LIN {X 0,Y 359.057,Z 1023.859,A -85,B 0,C 180,E1 26266.24,E2 26266.24} C_VEL
LIN {X 0,Y 361.976,Z 1017.878,A -85,B 0,C 180,E1 26267.168,E2 26267.168} C_VEL
LIN {X 0,Y 362.697,Z 1001.208,A -85,B 0,C 180,E1 26275.226,E2 26275.226} C_VEL
LIN {X 0,Y 363.155,Z 994.678,A -85,B 0,C 180,E1 26283.616,E2 26283.616} C_VEL
LIN {X 0,Y 361.753,Z 1005.173,A -85,B 0,C 180,E1 26293.358,E2 26293.358} C_VEL
LIN {X 0,Y 359.687,Z 1021.209,A -85,B 0,C 180,E1 26299.865,E2 26299.865} C_VEL
LIN {X 0,Y 316.249,Z 1080.703,A -85,B 0,C 180,E1 26305.848,E2 26305.848} C_VEL
LIN {X 0,Y 273.766,Z 1126.413,A -85,B 0,C 180,E1 26314.172,E2 26314.172} C_VEL
LIN {X 0,Y 249.213,Z 1145.042,A -85,B 0,C 180,E1 26318.032,E2 26318.032} C_VEL
LIN {X 0,Y 210.107,Z 1178.245,A -85,B 0,C 180,E1 26334.739,E2 26334.739} C_VEL
LIN {X 0,Y 190.164,Z 1197.047,A -85,B 0,C 180,E1 26356.165,E2 26356.165} C_VEL
LIN {X 0,Y 186.92,Z 1202.525,A -85,B 0,C 180,E1 26372.332,E2 26372.332} C_VEL
LIN {X 0,Y 188.619,Z 1200.708,A -85,B 0,C 180,E1 26392.237,E2 26392.237} C_VEL
LIN {X 0,Y 203.896,Z 1188.888,A -85,B 0,C 180,E1 26412.329,E2 26412.329} C_VEL
LIN {X 0,Y 242.392,Z 1161.787,A -85,B 0,C 180,E1 26431.043,E2 26431.043} C_VEL
LIN {X 0,Y 293.081,Z 1121.422,A -85,B 0,C 180,E1 26443.196,E2 26443.196} C_VEL
LIN {X 0,Y 345.638,Z 1068.573,A -85,B 0,C 180,E1 26450.834,E2 26450.834} C_VEL
LIN {X 0,Y 370.553,Z 1037.589,A -85,B 0,C 180,E1 26453.512,E2 26453.512} C_VEL
LIN {X 0,Y 372.422,Z 1029.57,A -85,B 0,C 180,E1 26461.144,E2 26461.144} C_VEL
LIN {X 0,Y 371.69,Z 1034.153,A -85,B 0,C 180,E1 26469.544,E2 26469.544} C_VEL
LIN {X 0,Y 369.889,Z 1039.513,A -85,B 0,C 180,E1 26472.259,E2 26472.259} C_VEL
LIN {X 0,Y 320.637,Z 1096.918,A -85,B 0,C 180,E1 26477.987,E2 26477.987} C_VEL
LIN {X 0,Y 267.811,Z 1144.547,A -85,B 0,C 180,E1 26487.487,E2 26487.487} C_VEL
LIN {X 0,Y 221.493,Z 1179.347,A -85,B 0,C 180,E1 26502.6,E2 26502.6} C_VEL
LIN {X 0,Y 193.031,Z 1200.435,A -85,B 0,C 180,E1 26524.393,E2 26524.393} C_VEL
LIN {X 0,Y 187.023,Z 1206.687,A -85,B 0,C 180,E1 26543.007,E2 26543.007} C_VEL
LIN {X 0,Y 187.02,Z 1205.903,A -85,B 0,C 180,E1 26556.979,E2 26556.979} C_VEL
LIN {X 0,Y 192.856,Z 1197.391,A -85,B 0,C 180,E1 26575.618,E2 26575.618} C_VEL
LIN {X 0,Y 218.915,Z 1173.79,A -85,B 0,C 180,E1 26596.656,E2 26596.656} C_VEL
LIN {X 0,Y 262.153,Z 1135.693,A -85,B 0,C 180,E1 26611.893,E2 26611.893} C_VEL
LIN {X 0,Y 311.561,Z 1084.366,A -85,B 0,C 180,E1 26621.632,E2 26621.632} C_VEL
LIN {X 0,Y 356.925,Z 1023.283,A -85,B 0,C 180,E1 26627.652,E2 26627.652} C_VEL
LIN {X 0,Y 358.203,Z 1006.363,A -85,B 0,C 180,E1 26636.382,E2 26636.382} C_VEL
LIN {X 0,Y 358.842,Z 1001.533,A -85,B 0,C 180,E1 26643.66,E2 26643.66} C_VEL
LIN {X 0,Y 357.045,Z 1012.278,A -85,B 0,C 180,E1 26653.538,E2 26653.538} C_VEL
LIN {X 0,Y 354.422,Z 1025.898,A -85,B 0,C 180,E1 26658.946,E2 26658.946} C_VEL
LIN {X 0,Y 308.073,Z 1086.636,A -85,B 0,C 180,E1 26665.255,E2 26665.255} C_VEL
LIN {X 0,Y 259.533,Z 1135.777,A -85,B 0,C 180,E1 26675.121,E2 26675.121} C_VEL
LIN {X 0,Y 249.213,Z 1145.042,A -85,B 0,C 180,E1 26678.032,E2 26678.032} C_VEL
LIN {X 0,Y 225.169,Z 1161.306,A -85,B 0,C 180,E1 26683.002,E2 26683.002} C_VEL
LIN {X 0,Y 192.438,Z 1187.662,A -85,B 0,C 180,E1 26701.79,E2 26701.79} C_VEL
LIN {X 0,Y 180.183,Z 1200.25,A -85,B 0,C 180,E1 26722.754,E2 26722.754} C_VEL
LIN {X 0,Y 178.43,Z 1202.977,A -85,B 0,C 180,E1 26737.331,E2 26737.331} C_VEL
LIN {X 0,Y 182.737,Z 1199.383,A -85,B 0,C 180,E1 26757.164,E2 26757.164} C_VEL
LIN {X 0,Y 205.467,Z 1183.588,A -85,B 0,C 180,E1 26779.28,E2 26779.28} C_VEL
LIN {X 0,Y 250.904,Z 1152.675,A -85,B 0,C 180,E1 26796.45,E2 26796.45} C_VEL
LIN {X 0,Y 305.086,Z 1108.368,A -85,B 0,C 180,E1 26807.14,E2 26807.14} C_VEL
LIN {X 0,Y 355.92,Z 1054.683,A -85,B 0,C 180,E1 26813.416,E2 26813.416} C_VEL
LIN {X 0,Y 365.792,Z 1042.038,A -85,B 0,C 180,E1 26814.623,E2 26814.623} C_VEL
LIN {X 0,Y 367.489,Z 1035.884,A -85,B 0,C 180,E1 26821.159,E2 26821.159} C_VEL
LIN {X 0,Y 366.523,Z 1040.357,A -85,B 0,C 180,E1 26829.505,E2 26829.505} C_VEL
LIN {X 0,Y 364.486,Z 1044.856,A -85,B 0,C 180,E1 26831.368,E2 26831.368} C_VEL
LIN {X 0,Y 314.252,Z 1101.025,A -85,B 0,C 180,E1 26837.107,E2 26837.107} C_VEL
LIN {X 0,Y 259.41,Z 1148.26,A -85,B 0,C 180,E1 26846.929,E2 26846.929} C_VEL
LIN {X 0,Y 212.09,Z 1181.955,A -85,B 0,C 180,E1 26862.744,E2 26862.744} C_VEL
LIN {X 0,Y 185.615,Z 1200.406,A -85,B 0,C 180,E1 26883.291,E2 26883.291} C_VEL
LIN {X 0,Y 179.014,Z 1206.607,A -85,B 0,C 180,E1 26902.693,E2 26902.693} C_VEL
LIN {X 0,Y 179.014,Z 1205.79,A -85,B 0,C 180,E1 26917.293,E2 26917.293} C_VEL
LIN {X 0,Y 185.425,Z 1197.223,A -85,B 0,C 180,E1 26936.724,E2 26936.724} C_VEL
LIN {X 0,Y 213.239,Z 1173.541,A -85,B 0,C 180,E1 26958.297,E2 26958.297} C_VEL
LIN {X 0,Y 258.302,Z 1135.348,A -85,B 0,C 180,E1 26973.537,E2 26973.537} C_VEL
LIN {X 0,Y 309.044,Z 1083.904,A -85,B 0,C 180,E1 26983.093,E2 26983.093} C_VEL
LIN {X 0,Y 352.115,Z 1026.928,A -85,B 0,C 180,E1 26988.847,E2 26988.847} C_VEL
LIN {X 0,Y 353.753,Z 1011.665,A -85,B 0,C 180,E1 26997.567,E2 26997.567} C_VEL
LIN {X 0,Y 354.286,Z 1008.235,A -85,B 0,C 180,E1 27003.707,E2 27003.707} C_VEL
LIN {X 0,Y 352.406,Z 1017.834,A -85,B 0,C 180,E1 27012.877,E2 27012.877} C_VEL
LIN {X 0,Y 349.886,Z 1029.624,A -85,B 0,C 180,E1 27017.931,E2 27017.931} C_VEL
LIN {X 0,Y 303.207,Z 1088.857,A -85,B 0,C 180,E1 27024.121,E2 27024.121} C_VEL
LIN {X 0,Y 252.35,Z 1138.513,A -85,B 0,C 180,E1 27034.29,E2 27034.29} C_VEL
LIN {X 0,Y 225.169,Z 1161.306,A -85,B 0,C 180,E1 27043.002,E2 27043.002} C_VEL
LIN {X 0,Y 201.919,Z 1175.08,A -85,B 0,C 180,E1 27049.206,E2 27049.206} C_VEL
LIN {X 0,Y 177.347,Z 1194.649,A -85,B 0,C 180,E1 27069.851,E2 27069.851} C_VEL
LIN {X 0,Y 171.336,Z 1201.777,A -85,B 0,C 180,E1 27087.471,E2 27087.471} C_VEL
LIN {X 0,Y 170.513,Z 1202.893,A -85,B 0,C 180,E1 27102.854,E2 27102.854} C_VEL
LIN {X 0,Y 180.26,Z 1196.11,A -85,B 0,C 180,E1 27125.586,E2 27125.586} C_VEL
LIN {X 0,Y 215.126,Z 1174.334,A -85,B 0,C 180,E1 27148.026,E2 27148.026} C_VEL
LIN {X 0,Y 267.617,Z 1137.874,A -85,B 0,C 180,E1 27162.694,E2 27162.694} C_VEL
LIN {X 0,Y 322.243,Z 1090.19,A -85,B 0,C 180,E1 27171.233,E2 27171.233} C_VEL
LIN {X 0,Y 360.885,Z 1047.179,A -85,B 0,C 180,E1 27175.393,E2 27175.393} C_VEL
LIN {X 0,Y 362.393,Z 1042.085,A -85,B 0,C 180,E1 27181.175,E2 27181.175} C_VEL
LIN {X 0,Y 361.335,Z 1046.614,A -85,B 0,C 180,E1 27189.49,E2 27189.49} C_VEL
LIN {X 0,Y 358.488,Z 1050.943,A -85,B 0,C 180,E1 27190.509,E2 27190.509} C_VEL
LIN {X 0,Y 306.352,Z 1106.665,A -85,B 0,C 180,E1 27196.435,E2 27196.435} C_VEL
LIN {X 0,Y 250.095,Z 1152.591,A -85,B 0,C 180,E1 27206.561,E2 27206.561} C_VEL
LIN {X 0,Y 203.168,Z 1184.206,A -85,B 0,C 180,E1 27222.649,E2 27222.649} C_VEL
LIN {X 0,Y 176.952,Z 1201.344,A -85,B 0,C 180,E1 27244.056,E2 27244.056} C_VEL
LIN {X 0,Y 171.034,Z 1206.527,A -85,B 0,C 180,E1 27262.35,E2 27262.35} C_VEL
LIN {X 0,Y 171.037,Z 1205.677,A -85,B 0,C 180,E1 27277.635,E2 27277.635} C_VEL
LIN {X 0,Y 179.966,Z 1195.448,A -85,B 0,C 180,E1 27300.362,E2 27300.362} C_VEL
LIN {X 0,Y 213.529,Z 1168.992,A -85,B 0,C 180,E1 27322.48,E2 27322.48} C_VEL
LIN {X 0,Y 260.468,Z 1130.014,A -85,B 0,C 180,E1 27336.476,E2 27336.476} C_VEL
LIN {X 0,Y 311.614,Z 1077.914,A -85,B 0,C 180,E1 27345.271,E2 27345.271} C_VEL
LIN {X 0,Y 347.033,Z 1032.286,A -85,B 0,C 180,E1 27349.463,E2 27349.463} C_VEL
LIN {X 0,Y 349.115,Z 1018.37,A -85,B 0,C 180,E1 27357.535,E2 27357.535} C_VEL
LIN {X 0,Y 349.734,Z 1014.931,A -85,B 0,C 180,E1 27363.755,E2 27363.755} C_VEL
LIN {X 0,Y 347.369,Z 1024.728,A -85,B 0,C 180,E1 27373.067,E2 27373.067} C_VEL
LIN {X 0,Y 345.026,Z 1033.835,A -85,B 0,C 180,E1 27376.93,E2 27376.93} C_VEL
LIN {X 0,Y 296.925,Z 1092.655,A -85,B 0,C 180,E1 27383.187,E2 27383.187} C_VEL
LIN {X 0,Y 245.221,Z 1141.031,A -85,B 0,C 180,E1 27393.409,E2 27393.409} C_VEL
LIN {X 0,Y 201.919,Z 1175.08,A -85,B 0,C 180,E1 27409.206,E2 27409.206} C_VEL
LIN {X 0,Y 181.003,Z 1186.16,A -85,B 0,C 180,E1 27417.17,E2 27417.17} C_VEL
LIN {X 0,Y 164.269,Z 1200.53,A -85,B 0,C 180,E1 27442.048,E2 27442.048} C_VEL
LIN {X 0,Y 162.3,Z 1203.134,A -85,B 0,C 180,E1 27460.807,E2 27460.807} C_VEL
LIN {X 0,Y 168.825,Z 1198.87,A -85,B 0,C 180,E1 27481.301,E2 27481.301} C_VEL
LIN {X 0,Y 198.533,Z 1181.376,A -85,B 0,C 180,E1 27504.985,E2 27504.985} C_VEL
LIN {X 0,Y 250.704,Z 1148.138,A -85,B 0,C 180,E1 27521.569,E2 27521.569} C_VEL
LIN {X 0,Y 307.506,Z 1102.666,A -85,B 0,C 180,E1 27531.092,E2 27531.092} C_VEL
LIN {X 0,Y 355.822,Z 1052.132,A -85,B 0,C 180,E1 27536.309,E2 27536.309} C_VEL
LIN {X 0,Y 357.27,Z 1048.377,A -85,B 0,C 180,E1 27544.024,E2 27544.024} C_VEL
LIN {X 0,Y 355.197,Z 1053.542,A -85,B 0,C 180,E1 27549.396,E2 27549.396} C_VEL
LIN {X 0,Y 302.464,Z 1108.331,A -85,B 0,C 180,E1 27555.159,E2 27555.159} C_VEL
LIN {X 0,Y 246.487,Z 1152.707,A -85,B 0,C 180,E1 27564.831,E2 27564.831} C_VEL
LIN {X 0,Y 196.592,Z 1184.795,A -85,B 0,C 180,E1 27581.349,E2 27581.349} C_VEL
LIN {X 0,Y 167.651,Z 1202.71,A -85,B 0,C 180,E1 27605.973,E2 27605.973} C_VEL
LIN {X 0,Y 162.931,Z 1206.761,A -85,B 0,C 180,E1 27627.325,E2 27627.325} C_VEL
LIN {X 0,Y 163.788,Z 1204.118,A -85,B 0,C 180,E1 27643.714,E2 27643.714} C_VEL
LIN {X 0,Y 178.266,Z 1191.028,A -85,B 0,C 180,E1 27667.032,E2 27667.032} C_VEL
LIN {X 0,Y 216.194,Z 1162.786,A -85,B 0,C 180,E1 27687.311,E2 27687.311} C_VEL
LIN {X 0,Y 266.24,Z 1121.478,A -85,B 0,C 180,E1 27700.006,E2 27700.006} C_VEL
LIN {X 0,Y 317.99,Z 1067.573,A -85,B 0,C 180,E1 27707.837,E2 27707.837} C_VEL
LIN {X 0,Y 342.342,Z 1035.885,A -85,B 0,C 180,E1 27710.723,E2 27710.723} C_VEL
LIN {X 0,Y 344.651,Z 1022.943,A -85,B 0,C 180,E1 27719.534,E2 27719.534} C_VEL
LIN {X 0,Y 344.959,Z 1021.491,A -85,B 0,C 180,E1 27723.807,E2 27723.807} C_VEL
LIN {X 0,Y 342.447,Z 1030.894,A -85,B 0,C 180,E1 27732.822,E2 27732.822} C_VEL
LIN {X 0,Y 340.239,Z 1037.865,A -85,B 0,C 180,E1 27735.907,E2 27735.907} C_VEL
LIN {X 0,Y 290.704,Z 1096.259,A -85,B 0,C 180,E1 27742.203,E2 27742.203} C_VEL
LIN {X 0,Y 237.304,Z 1144.175,A -85,B 0,C 180,E1 27752.689,E2 27752.689} C_VEL
LIN {X 0,Y 192.465,Z 1177.693,A -85,B 0,C 180,E1 27769.465,E2 27769.465} C_VEL
LIN {X 0,Y 181.003,Z 1186.16,A -85,B 0,C 180,E1 27777.17,E2 27777.17} C_VEL
LIN {X 0,Y 162.839,Z 1194.5,A -85,B 0,C 180,E1 27786.993,E2 27786.993} C_VEL
LIN {X 0,Y 155.347,Z 1202.014,A -85,B 0,C 180,E1 27807.21,E2 27807.21} C_VEL
LIN {X 0,Y 154.584,Z 1203.051,A -85,B 0,C 180,E1 27824.205,E2 27824.205} C_VEL
LIN {X 0,Y 167.097,Z 1195.881,A -85,B 0,C 180,E1 27849.42,E2 27849.42} C_VEL
LIN {X 0,Y 206.857,Z 1173.856,A -85,B 0,C 180,E1 27872.308,E2 27872.308} C_VEL
LIN {X 0,Y 262.577,Z 1137.78,A -85,B 0,C 180,E1 27886.219,E2 27886.219} C_VEL
LIN {X 0,Y 320.915,Z 1088.688,A -85,B 0,C 180,E1 27894.36,E2 27894.36} C_VEL
LIN {X 0,Y 350.797,Z 1056.986,A -85,B 0,C 180,E1 27897.362,E2 27897.362} C_VEL
LIN {X 0,Y 352.028,Z 1054.19,A -85,B 0,C 180,E1 27903.681,E2 27903.681} C_VEL
LIN {X 0,Y 349.905,Z 1058.636,A -85,B 0,C 180,E1 27908.44,E2 27908.44} C_VEL
LIN {X 0,Y 293.69,Z 1114.329,A -85,B 0,C 180,E1 27914.483,E2 27914.483} C_VEL
LIN {X 0,Y 235.649,Z 1157.721,A -85,B 0,C 180,E1 27924.693,E2 27924.693} C_VEL
LIN {X 0,Y 185.157,Z 1188.174,A -85,B 0,C 180,E1 27942.504,E2 27942.504} C_VEL
LIN {X 0,Y 160.164,Z 1202.663,A -85,B 0,C 180,E1 27964.773,E2 27964.773} C_VEL
LIN {X 0,Y 154.916,Z 1206.664,A -85,B 0,C 180,E1 27987.186,E2 27987.186} C_VEL
LIN {X 0,Y 155.858,Z 1204.096,A -85,B 0,C 180,E1 28004.07,E2 28004.07} C_VEL
LIN {X 0,Y 172.672,Z 1190.17,A -85,B 0,C 180,E1 28029.538,E2 28029.538} C_VEL
LIN {X 0,Y 214.306,Z 1160.693,A -85,B 0,C 180,E1 28050.075,E2 28050.075} C_VEL
LIN {X 0,Y 268.216,Z 1116.843,A -85,B 0,C 180,E1 28062.556,E2 28062.556} C_VEL
LIN {X 0,Y 321.241,Z 1061.179,A -85,B 0,C 180,E1 28069.862,E2 28069.862} C_VEL
LIN {X 0,Y 337.452,Z 1040.055,A -85,B 0,C 180,E1 28071.816,E2 28071.816} C_VEL
LIN {X 0,Y 340.008,Z 1028.718,A -85,B 0,C 180,E1 28080.415,E2 28080.415} C_VEL
LIN {X 0,Y 339.016,Z 1030.447,A -85,B 0,C 180,E1 28087.321,E2 28087.321} C_VEL
LIN {X 0,Y 336.521,Z 1040.103,A -85,B 0,C 180,E1 28094.381,E2 28094.381} C_VEL
LIN {X 0,Y 289.144,Z 1095.339,A -85,B 0,C 180,E1 28100.509,E2 28100.509} C_VEL
LIN {X 0,Y 235.092,Z 1142.915,A -85,B 0,C 180,E1 28110.49,E2 28110.49} C_VEL
LIN {X 0,Y 188.273,Z 1176.636,A -85,B 0,C 180,E1 28126.802,E2 28126.802} C_VEL
LIN {X 0,Y 162.839,Z 1194.5,A -85,B 0,C 180,E1 28146.993,E2 28146.993} C_VEL
LIN {X 0,Y 148.901,Z 1200.112,A -85,B 0,C 180,E1 28158.881,E2 28158.881} C_VEL
LIN {X 0,Y 146.292,Z 1203.409,A -85,B 0,C 180,E1 28179.578,E2 28179.578} C_VEL
LIN {X 0,Y 155.531,Z 1198.376,A -85,B 0,C 180,E1 28205.814,E2 28205.814} C_VEL
LIN {X 0,Y 191.905,Z 1179.73,A -85,B 0,C 180,E1 28230.383,E2 28230.383} C_VEL
LIN {X 0,Y 248.295,Z 1146.082,A -85,B 0,C 180,E1 28245.865,E2 28245.865} C_VEL
LIN {X 0,Y 307.204,Z 1100.364,A -85,B 0,C 180,E1 28254.483,E2 28254.483} C_VEL
LIN {X 0,Y 345.752,Z 1062.062,A -85,B 0,C 180,E1 28258.305,E2 28258.305} C_VEL
LIN {X 0,Y 346.629,Z 1060.197,A -85,B 0,C 180,E1 28263.738,E2 28263.738} C_VEL
LIN {X 0,Y 345.806,Z 1062.402,A -85,B 0,C 180,E1 28267.251,E2 28267.251} C_VEL
LIN {X 0,Y 287.064,Z 1118.52,A -85,B 0,C 180,E1 28273.508,E2 28273.508} C_VEL
LIN {X 0,Y 226.827,Z 1161.34,A -85,B 0,C 180,E1 28284.083,E2 28284.083} C_VEL
LIN {X 0,Y 175.551,Z 1190.382,A -85,B 0,C 180,E1 28302.745,E2 28302.745} C_VEL
LIN {X 0,Y 149.793,Z 1204.366,A -85,B 0,C 180,E1 28329.239,E2 28329.239} C_VEL
LIN {X 0,Y 146.895,Z 1206.568,A -85,B 0,C 180,E1 28347.033,E2 28347.033} C_VEL
LIN {X 0,Y 148.008,Z 1203.964,A -85,B 0,C 180,E1 28364.833,E2 28364.833} C_VEL
LIN {X 0,Y 166.289,Z 1189.973,A -85,B 0,C 180,E1 28391.378,E2 28391.378} C_VEL
LIN {X 0,Y 210.286,Z 1160.348,A -85,B 0,C 180,E1 28412.086,E2 28412.086} C_VEL
LIN {X 0,Y 265.803,Z 1116.432,A -85,B 0,C 180,E1 28424.295,E2 28424.295} C_VEL
LIN {X 0,Y 319.415,Z 1061.188,A -85,B 0,C 180,E1 28431.29,E2 28431.29} C_VEL
LIN {X 0,Y 332.628,Z 1044.33,A -85,B 0,C 180,E1 28432.913,E2 28432.913} C_VEL
LIN {X 0,Y 335.402,Z 1034.441,A -85,B 0,C 180,E1 28441.322,E2 28441.322} C_VEL
LIN {X 0,Y 333.401,Z 1038.582,A -85,B 0,C 180,E1 28449.189,E2 28449.189} C_VEL
LIN {X 0,Y 330.188,Z 1047.027,A -85,B 0,C 180,E1 28453.874,E2 28453.874} C_VEL
LIN {X 0,Y 278.219,Z 1103.775,A -85,B 0,C 180,E1 28460.152,E2 28460.152} C_VEL
LIN {X 0,Y 223.199,Z 1149.229,A -85,B 0,C 180,E1 28470.689,E2 28470.689} C_VEL
LIN {X 0,Y 174.646,Z 1182.003,A -85,B 0,C 180,E1 28489.375,E2 28489.375} C_VEL
LIN {X 0,Y 150.122,Z 1199.043,A -85,B 0,C 180,E1 28515.381,E2 28515.381} C_VEL
LIN {X 0,Y 148.901,Z 1200.112,A -85,B 0,C 180,E1 28518.881,E2 28518.881} C_VEL
LIN {X 0,Y 138.658,Z 1203.028,A -85,B 0,C 180,E1 28532.51,E2 28532.51} C_VEL
LIN {X 0,Y 142.722,Z 1201.284,A -85,B 0,C 180,E1 28558.574,E2 28558.574} C_VEL
LIN {X 0,Y 169.218,Z 1188.684,A -85,B 0,C 180,E1 28584.299,E2 28584.299} C_VEL
LIN {X 0,Y 222.075,Z 1160.936,A -85,B 0,C 180,E1 28602.953,E2 28602.953} C_VEL
LIN {X 0,Y 284.231,Z 1118.711,A -85,B 0,C 180,E1 28613.512,E2 28613.512} C_VEL
LIN {X 0,Y 340.485,Z 1067.147,A -85,B 0,C 180,E1 28619.336,E2 28619.336} C_VEL
LIN {X 0,Y 340.472,Z 1067.539,A -85,B 0,C 180,E1 28626.369,E2 28626.369} C_VEL
LIN {X 0,Y 283.938,Z 1119.718,A -85,B 0,C 180,E1 28632.05,E2 28632.05} C_VEL
LIN {X 0,Y 221.685,Z 1162.503,A -85,B 0,C 180,E1 28642.545,E2 28642.545} C_VEL
LIN {X 0,Y 169.992,Z 1190.393,A -85,B 0,C 180,E1 28660.677,E2 28660.677} C_VEL
LIN {X 0,Y 142.159,Z 1204.32,A -85,B 0,C 180,E1 28688.068,E2 28688.068} C_VEL
LIN {X 0,Y 138.892,Z 1206.472,A -85,B 0,C 180,E1 28706.862,E2 28706.862} C_VEL
LIN {X 0,Y 140.147,Z 1203.832,A -85,B 0,C 180,E1 28725.685,E2 28725.685} C_VEL
LIN {X 0,Y 160.098,Z 1189.768,A -85,B 0,C 180,E1 28753.361,E2 28753.361} C_VEL
LIN {X 0,Y 205.773,Z 1160.533,A -85,B 0,C 180,E1 28773.966,E2 28773.966} C_VEL
LIN {X 0,Y 261.809,Z 1117.68,A -85,B 0,C 180,E1 28785.768,E2 28785.768} C_VEL
LIN {X 0,Y 316.112,Z 1063.227,A -85,B 0,C 180,E1 28792.56,E2 28792.56} C_VEL
LIN {X 0,Y 327.791,Z 1048.78,A -85,B 0,C 180,E1 28794.036,E2 28794.036} C_VEL
LIN {X 0,Y 330.294,Z 1040.651,A -85,B 0,C 180,E1 28801.342,E2 28801.342} C_VEL
LIN {X 0,Y 328.157,Z 1045.04,A -85,B 0,C 180,E1 28809.337,E2 28809.337} C_VEL
LIN {X 0,Y 325.883,Z 1050.637,A -85,B 0,C 180,E1 28812.74,E2 28812.74} C_VEL
LIN {X 0,Y 272.596,Z 1106.842,A -85,B 0,C 180,E1 28818.98,E2 28818.98} C_VEL
LIN {X 0,Y 217.349,Z 1150.776,A -85,B 0,C 180,E1 28829.304,E2 28829.304} C_VEL
LIN {X 0,Y 168.531,Z 1182.229,A -85,B 0,C 180,E1 28847.567,E2 28847.567} C_VEL
LIN {X 0,Y 142.364,Z 1199.204,A -85,B 0,C 180,E1 28874.565,E2 28874.565} C_VEL
LIN {X 0,Y 138.658,Z 1203.028,A -85,B 0,C 180,E1 28892.51,E2 28892.51} C_VEL
LIN {X 0,Y 130.886,Z 1203.237,A -85,B 0,C 180,E1 28907.33,E2 28907.33} C_VEL
LIN {X 0,Y 148.145,Z 1195.852,A -85,B 0,C 180,E1 28935.782,E2 28935.782} C_VEL
LIN {X 0,Y 196.33,Z 1173.428,A -85,B 0,C 180,E1 28959.168,E2 28959.168} C_VEL
LIN {X 0,Y 257.14,Z 1137.517,A -85,B 0,C 180,E1 28971.767,E2 28971.767} C_VEL
LIN {X 0,Y 318.79,Z 1088.315,A -85,B 0,C 180,E1 28978.885,E2 28978.885} C_VEL
LIN {X 0,Y 335.16,Z 1072.266,A -85,B 0,C 180,E1 28980.4,E2 28980.4} C_VEL
LIN {X 0,Y 335.071,Z 1072.574,A -85,B 0,C 180,E1 28985.17,E2 28985.17} C_VEL
LIN {X 0,Y 274.156,Z 1126.091,A -85,B 0,C 180,E1 28991.377,E2 28991.377} C_VEL
LIN {X 0,Y 212.515,Z 1166.05,A -85,B 0,C 180,E1 29001.913,E2 29001.913} C_VEL
LIN {X 0,Y 159.817,Z 1192.596,A -85,B 0,C 180,E1 29021.171,E2 29021.171} C_VEL
LIN {X 0,Y 134.595,Z 1204.274,A -85,B 0,C 180,E1 29046.765,E2 29046.765} C_VEL
LIN {X 0,Y 130.869,Z 1206.375,A -85,B 0,C 180,E1 29066.669,E2 29066.669} C_VEL
LIN {X 0,Y 132.338,Z 1203.699,A -85,B 0,C 180,E1 29086.637,E2 29086.637} C_VEL
LIN {X 0,Y 154.083,Z 1189.556,A -85,B 0,C 180,E1 29115.511,E2 29115.511} C_VEL
LIN {X 0,Y 202.186,Z 1160.248,A -85,B 0,C 180,E1 29136.107,E2 29136.107} C_VEL
LIN {X 0,Y 260.403,Z 1116.782,A -85,B 0,C 180,E1 29147.659,E2 29147.659} C_VEL
LIN {X 0,Y 315.895,Z 1061.766,A -85,B 0,C 180,E1 29154.149,E2 29154.149} C_VEL
LIN {X 0,Y 322.85,Z 1053.088,A -85,B 0,C 180,E1 29155.256,E2 29155.256} C_VEL
LIN {X 0,Y 325.17,Z 1046.88,A -85,B 0,C 180,E1 29161.363,E2 29161.363} C_VEL
LIN {X 0,Y 322.748,Z 1051.423,A -85,B 0,C 180,E1 29169.495,E2 29169.495} C_VEL
LIN {X 0,Y 320.396,Z 1055.693,A -85,B 0,C 180,E1 29171.701,E2 29171.701} C_VEL
LIN {X 0,Y 265.113,Z 1111.563,A -85,B 0,C 180,E1 29178.034,E2 29178.034} C_VEL
LIN {X 0,Y 207,Z 1155.412,A -85,B 0,C 180,E1 29189.05,E2 29189.05} C_VEL
LIN {X 0,Y 156.75,Z 1185.823,A -85,B 0,C 180,E1 29209.241,E2 29209.241} C_VEL
LIN {X 0,Y 134.629,Z 1199.364,A -85,B 0,C 180,E1 29233.654,E2 29233.654} C_VEL
LIN {X 0,Y 130.605,Z 1203.214,A -85,B 0,C 180,E1 29253.338,E2 29253.338} C_VEL
LIN {X 0,Y 130.886,Z 1203.237,A -85,B 0,C 180,E1 29267.33,E2 29267.33} C_VEL
LIN {X 0,Y 128.668,Z 1201.154,A -85,B 0,C 180,E1 29283.003,E2 29283.003} C_VEL
LIN {X 0,Y 164.13,Z 1186.796,A -85,B 0,C 180,E1 29311.387,E2 29311.387} C_VEL
LIN {X 0,Y 224.324,Z 1156.923,A -85,B 0,C 180,E1 29328.612,E2 29328.612} C_VEL
LIN {X 0,Y 288.409,Z 1113.843,A -85,B 0,C 180,E1 29337.565,E2 29337.565} C_VEL
LIN {X 0,Y 329.846,Z 1077.514,A -85,B 0,C 180,E1 29341.291,E2 29341.291} C_VEL
LIN {X 0,Y 329.011,Z 1078.501,A -85,B 0,C 180,E1 29344.354,E2 29344.354} C_VEL
LIN {X 0,Y 266.043,Z 1131.119,A -85,B 0,C 180,E1 29350.474,E2 29350.474} C_VEL
LIN {X 0,Y 203.364,Z 1169.522,A -85,B 0,C 180,E1 29361.218,E2 29361.218} C_VEL
LIN {X 0,Y 150.767,Z 1194.272,A -85,B 0,C 180,E1 29381.017,E2 29381.017} C_VEL
LIN {X 0,Y 124.503,Z 1205.363,A -85,B 0,C 180,E1 29412.261,E2 29412.261} C_VEL
LIN {X 0,Y 122.841,Z 1205.942,A -85,B 0,C 180,E1 29433.529,E2 29433.529} C_VEL
LIN {X 0,Y 130.918,Z 1199.167,A -85,B 0,C 180,E1 29461.405,E2 29461.405} C_VEL
LIN {X 0,Y 168.912,Z 1177.91,A -85,B 0,C 180,E1 29488.513,E2 29488.513} C_VEL
LIN {X 0,Y 226.368,Z 1141.474,A -85,B 0,C 180,E1 29504.343,E2 29504.343} C_VEL
LIN {X 0,Y 286.541,Z 1091.36,A -85,B 0,C 180,E1 29512.852,E2 29512.852} C_VEL
LIN {X 0,Y 317.615,Z 1058.283,A -85,B 0,C 180,E1 29515.919,E2 29515.919} C_VEL
LIN {X 0,Y 319.865,Z 1052.95,A -85,B 0,C 180,E1 29521.386,E2 29521.386} C_VEL
LIN {X 0,Y 317.193,Z 1057.669,A -85,B 0,C 180,E1 29529.663,E2 29529.663} C_VEL
LIN {X 0,Y 314.064,Z 1061.864,A -85,B 0,C 180,E1 29530.717,E2 29530.717} C_VEL
LIN {X 0,Y 257.7,Z 1116.292,A -85,B 0,C 180,E1 29537.039,E2 29537.039} C_VEL
LIN {X 0,Y 198.129,Z 1159.025,A -85,B 0,C 180,E1 29548.347,E2 29548.347} C_VEL
LIN {X 0,Y 148.737,Z 1187.172,A -85,B 0,C 180,E1 29568.504,E2 29568.504} C_VEL
LIN {X 0,Y 124.685,Z 1201.225,A -85,B 0,C 180,E1 29599.499,E2 29599.499} C_VEL
LIN {X 0,Y 122.261,Z 1203.671,A -85,B 0,C 180,E1 29620.733,E2 29620.733} C_VEL
LIN {X 0,Y 128.668,Z 1201.154,A -85,B 0,C 180,E1 29643.003,E2 29643.003} C_VEL
LIN {X 0,Y 133.466,Z 1197.027,A -85,B 0,C 180,E1 29658.369,E2 29658.369} C_VEL
LIN {X 0,Y 186.334,Z 1175.433,A -85,B 0,C 180,E1 29682.856,E2 29682.856} C_VEL
LIN {X 0,Y 251.166,Z 1139.869,A -85,B 0,C 180,E1 29695.071,E2 29695.071} C_VEL
LIN {X 0,Y 314.805,Z 1091.497,A -85,B 0,C 180,E1 29701.624,E2 29701.624} C_VEL
LIN {X 0,Y 323.906,Z 1083.048,A -85,B 0,C 180,E1 29702.657,E2 29702.657} C_VEL
LIN {X 0,Y 320.402,Z 1086.358,A -85,B 0,C 180,E1 29703.508,E2 29703.508} C_VEL
LIN {X 0,Y 257.613,Z 1136.056,A -85,B 0,C 180,E1 29709.569,E2 29709.569} C_VEL
LIN {X 0,Y 193.623,Z 1172.948,A -85,B 0,C 180,E1 29720.594,E2 29720.594} C_VEL
LIN {X 0,Y 141.152,Z 1195.894,A -85,B 0,C 180,E1 29741.219,E2 29741.219} C_VEL
LIN {X 0,Y 116.771,Z 1205.3,A -85,B 0,C 180,E1 29771.043,E2 29771.043} C_VEL
LIN {X 0,Y 114.818,Z 1205.845,A -85,B 0,C 180,E1 29793.776,E2 29793.776} C_VEL
LIN {X 0,Y 123.934,Z 1199.013,A -85,B 0,C 180,E1 29823.397,E2 29823.397} C_VEL
LIN {X 0,Y 164.695,Z 1177.675,A -85,B 0,C 180,E1 29850.997,E2 29850.997} C_VEL
LIN {X 0,Y 223.719,Z 1141.498,A -85,B 0,C 180,E1 29866.312,E2 29866.312} C_VEL
LIN {X 0,Y 283.804,Z 1092.669,A -85,B 0,C 180,E1 29874.335,E2 29874.335} C_VEL
LIN {X 0,Y 312.721,Z 1062.706,A -85,B 0,C 180,E1 29877.246,E2 29877.246} C_VEL
LIN {X 0,Y 314.466,Z 1058.938,A -85,B 0,C 180,E1 29881.41,E2 29881.41} C_VEL
LIN {X 0,Y 312.002,Z 1063.005,A -85,B 0,C 180,E1 29889.01,E2 29889.01} C_VEL
LIN {X 0,Y 256.53,Z 1115.797,A -85,B 0,C 180,E1 29895.157,E2 29895.157} C_VEL
LIN {X 0,Y 196.094,Z 1158.266,A -85,B 0,C 180,E1 29905.8,E2 29905.8} C_VEL
LIN {X 0,Y 142.736,Z 1187.394,A -85,B 0,C 180,E1 29926.337,E2 29926.337} C_VEL
LIN {X 0,Y 116.798,Z 1201.364,A -85,B 0,C 180,E1 29958.781,E2 29958.781} C_VEL
LIN {X 0,Y 114.261,Z 1203.764,A -85,B 0,C 180,E1 29981.494,E2 29981.494} C_VEL
LIN {X 0,Y 128.741,Z 1198.716,A -85,B 0,C 180,E1 30013.932,E2 30013.932} C_VEL
LIN {X 0,Y 133.466,Z 1197.027,A -85,B 0,C 180,E1 30018.369,E2 30018.369} C_VEL
LIN {X 0,Y 145.078,Z 1190.973,A -85,B 0,C 180,E1 30031.993,E2 30031.993} C_VEL
LIN {X 0,Y 207.535,Z 1163.985,A -85,B 0,C 180,E1 30050.593,E2 30050.593} C_VEL
LIN {X 0,Y 275.09,Z 1123.043,A -85,B 0,C 180,E1 30059.76,E2 30059.76} C_VEL
LIN {X 0,Y 308.545,Z 1096.853,A -85,B 0,C 180,E1 30062.877,E2 30062.877} C_VEL
LIN {X 0,Y 243.224,Z 1144.615,A -85,B 0,C 180,E1 30069.336,E2 30069.336} C_VEL
LIN {X 0,Y 175.952,Z 1179.857,A -85,B 0,C 180,E1 30082.085,E2 30082.085} C_VEL
LIN {X 0,Y 123.738,Z 1200.152,A -85,B 0,C 180,E1 30107.606,E2 30107.606} C_VEL
LIN {X 0,Y 107.301,Z 1205.888,A -85,B 0,C 180,E1 30137.749,E2 30137.749} C_VEL
LIN {X 0,Y 107.317,Z 1204.764,A -85,B 0,C 180,E1 30162.225,E2 30162.225} C_VEL
LIN {X 0,Y 127.152,Z 1193.958,A -85,B 0,C 180,E1 30195.677,E2 30195.677} C_VEL
LIN {X 0,Y 178.354,Z 1167.957,A -85,B 0,C 180,E1 30219.253,E2 30219.253} C_VEL
LIN {X 0,Y 239.643,Z 1128.455,A -85,B 0,C 180,E1 30231.06,E2 30231.06} C_VEL
LIN {X 0,Y 298.965,Z 1076.591,A -85,B 0,C 180,E1 30237.469,E2 30237.469} C_VEL
LIN {X 0,Y 307.724,Z 1067.157,A -85,B 0,C 180,E1 30238.616,E2 30238.616} C_VEL
LIN {X 0,Y 308.582,Z 1065.15,A -85,B 0,C 180,E1 30244.257,E2 30244.257} C_VEL
LIN {X 0,Y 305.334,Z 1069.464,A -85,B 0,C 180,E1 30248.311,E2 30248.311} C_VEL
LIN {X 0,Y 246.46,Z 1122.42,A -85,B 0,C 180,E1 30254.391,E2 30254.391} C_VEL
LIN {X 0,Y 184.839,Z 1163.012,A -85,B 0,C 180,E1 30265.532,E2 30265.532} C_VEL
LIN {X 0,Y 132.713,Z 1189.497,A -85,B 0,C 180,E1 30286.73,E2 30286.73} C_VEL
LIN {X 0,Y 108.936,Z 1201.502,A -85,B 0,C 180,E1 30317.959,E2 30317.959} C_VEL
LIN {X 0,Y 106.259,Z 1203.85,A -85,B 0,C 180,E1 30342.373,E2 30342.373} C_VEL
LIN {X 0,Y 123.477,Z 1198.484,A -85,B 0,C 180,E1 30377.4,E2 30377.4} C_VEL
LIN {X 0,Y 145.078,Z 1190.973,A -85,B 0,C 180,E1 30391.993,E2 30391.993} C_VEL
LIN {X 0,Y 163.121,Z 1183.007,A -85,B 0,C 180,E1 30403.024,E2 30403.024} C_VEL
LIN {X 0,Y 229.398,Z 1151.772,A -85,B 0,C 180,E1 30416.445,E2 30416.445} C_VEL
LIN {X 0,Y 288.632,Z 1112.963,A -85,B 0,C 180,E1 30422.828,E2 30422.828} C_VEL
LIN {X 0,Y 223.188,Z 1155.616,A -85,B 0,C 180,E1 30429.835,E2 30429.835} C_VEL
LIN {X 0,Y 155.154,Z 1187.107,A -85,B 0,C 180,E1 30444.863,E2 30444.863} C_VEL
LIN {X 0,Y 110.711,Z 1202.344,A -85,B 0,C 180,E1 30471.933,E2 30471.933} C_VEL
LIN {X 0,Y 98.811,Z 1205.989,A -85,B 0,C 180,E1 30505.586,E2 30505.586} C_VEL
LIN {X 0,Y 101.476,Z 1203.164,A -85,B 0,C 180,E1 30531.925,E2 30531.925} C_VEL
LIN {X 0,Y 131.626,Z 1189.208,A -85,B 0,C 180,E1 30565.339,E2 30565.339} C_VEL
LIN {X 0,Y 188.429,Z 1160.527,A -85,B 0,C 180,E1 30584.935,E2 30584.935} C_VEL
LIN {X 0,Y 251.3,Z 1118.401,A -85,B 0,C 180,E1 30594.622,E2 30594.622} C_VEL
LIN {X 0,Y 302.509,Z 1071.992,A -85,B 0,C 180,E1 30599.676,E2 30599.676} C_VEL
LIN {X 0,Y 302.098,Z 1071.924,A -85,B 0,C 180,E1 30605.77,E2 30605.77} C_VEL
LIN {X 0,Y 299.563,Z 1074.865,A -85,B 0,C 180,E1 30607.174,E2 30607.174} C_VEL
LIN {X 0,Y 239.439,Z 1126.654,A -85,B 0,C 180,E1 30613.179,E2 30613.179} C_VEL
LIN {X 0,Y 178.375,Z 1165.005,A -85,B 0,C 180,E1 30623.966,E2 30623.966} C_VEL
LIN {X 0,Y 122.638,Z 1191.585,A -85,B 0,C 180,E1 30647.163,E2 30647.163} C_VEL
LIN {X 0,Y 100.396,Z 1202.134,A -85,B 0,C 180,E1 30679.602,E2 30679.602} C_VEL
LIN {X 0,Y 98.292,Z 1203.93,A -85,B 0,C 180,E1 30703.394,E2 30703.394} C_VEL
LIN {X 0,Y 117.841,Z 1198.504,A -85,B 0,C 180,E1 30740.47,E2 30740.47} C_VEL
LIN {X 0,Y 163.121,Z 1183.007,A -85,B 0,C 180,E1 30763.024,E2 30763.024} C_VEL
LIN {X 0,Y 184.769,Z 1173.222,A -85,B 0,C 180,E1 30771.75,E2 30771.75} C_VEL
LIN {X 0,Y 255.837,Z 1135.739,A -85,B 0,C 180,E1 30781.557,E2 30781.557} C_VEL
LIN {X 0,Y 268.387,Z 1127.594,A -85,B 0,C 180,E1 30782.721,E2 30782.721} C_VEL
LIN {X 0,Y 196.84,Z 1168.462,A -85,B 0,C 180,E1 30791.408,E2 30791.408} C_VEL
LIN {X 0,Y 131.259,Z 1194.303,A -85,B 0,C 180,E1 30809.928,E2 30809.928} C_VEL
LIN {X 0,Y 93.912,Z 1205.113,A -85,B 0,C 180,E1 30846.176,E2 30846.176} C_VEL
LIN {X 0,Y 90.822,Z 1205.555,A -85,B 0,C 180,E1 30874.775,E2 30874.775} C_VEL
LIN {X 0,Y 107.045,Z 1197.236,A -85,B 0,C 180,E1 30914.031,E2 30914.031} C_VEL
LIN {X 0,Y 159.273,Z 1174.359,A -85,B 0,C 180,E1 30940.827,E2 30940.827} C_VEL
LIN {X 0,Y 224.072,Z 1137.063,A -85,B 0,C 180,E1 30953.429,E2 30953.429} C_VEL
LIN {X 0,Y 287.024,Z 1086.851,A -85,B 0,C 180,E1 30959.791,E2 30959.791} C_VEL
LIN {X 0,Y 297.317,Z 1076.916,A -85,B 0,C 180,E1 30960.764,E2 30960.764} C_VEL
LIN {X 0,Y 296.483,Z 1077.593,A -85,B 0,C 180,E1 30965.649,E2 30965.649} C_VEL
LIN {X 0,Y 234.202,Z 1129.593,A -85,B 0,C 180,E1 30971.693,E2 30971.693} C_VEL
LIN {X 0,Y 168.971,Z 1168.548,A -85,B 0,C 180,E1 30983.046,E2 30983.046} C_VEL
LIN {X 0,Y 113.11,Z 1193.273,A -85,B 0,C 180,E1 31007.181,E2 31007.181} C_VEL
LIN {X 0,Y 91.459,Z 1202.957,A -85,B 0,C 180,E1 31045.258,E2 31045.258} C_VEL
LIN {X 0,Y 92.299,Z 1203.664,A -85,B 0,C 180,E1 31075.106,E2 31075.106} C_VEL
LIN {X 0,Y 122.579,Z 1195.662,A -85,B 0,C 180,E1 31110.827,E2 31110.827} C_VEL
LIN {X 0,Y 184.769,Z 1173.222,A -85,B 0,C 180,E1 31131.75,E2 31131.75} C_VEL
LIN {X 0,Y 209.381,Z 1161.528,A -85,B 0,C 180,E1 31138.39,E2 31138.39} C_VEL
LIN {X 0,Y 245.673,Z 1142.022,A -85,B 0,C 180,E1 31142.518,E2 31142.518} C_VEL
LIN {X 0,Y 176.197,Z 1176.845,A -85,B 0,C 180,E1 31152.378,E2 31152.378} C_VEL
LIN {X 0,Y 111.399,Z 1198.855,A -85,B 0,C 180,E1 31175.218,E2 31175.218} C_VEL
LIN {X 0,Y 83.678,Z 1205.649,A -85,B 0,C 180,E1 31214.211,E2 31214.211} C_VEL
LIN {X 0,Y 82.809,Z 1205.455,A -85,B 0,C 180,E1 31235.238,E2 31235.238} C_VEL
LIN {X 0,Y 98.004,Z 1198.37,A -85,B 0,C 180,E1 31274.113,E2 31274.113} C_VEL
LIN {X 0,Y 151.268,Z 1176.719,A -85,B 0,C 180,E1 31302.218,E2 31302.218} C_VEL
LIN {X 0,Y 217.559,Z 1140.549,A -85,B 0,C 180,E1 31314.851,E2 31314.851} C_VEL
LIN {X 0,Y 282.451,Z 1090.742,A -85,B 0,C 180,E1 31321.141,E2 31321.141} C_VEL
LIN {X 0,Y 291.681,Z 1082.021,A -85,B 0,C 180,E1 31322.265,E2 31322.265} C_VEL
LIN {X 0,Y 290.221,Z 1083.335,A -85,B 0,C 180,E1 31324.639,E2 31324.639} C_VEL
LIN {X 0,Y 227.163,Z 1133.612,A -85,B 0,C 180,E1 31330.347,E2 31330.347} C_VEL
LIN {X 0,Y 159.473,Z 1171.849,A -85,B 0,C 180,E1 31342.027,E2 31342.027} C_VEL
LIN {X 0,Y 102.366,Z 1195.202,A -85,B 0,C 180,E1 31368.209,E2 31368.209} C_VEL
LIN {X 0,Y 83.478,Z 1203.074,A -85,B 0,C 180,E1 31404.804,E2 31404.804} C_VEL
LIN {X 0,Y 84.612,Z 1203.77,A -85,B 0,C 180,E1 31436.636,E2 31436.636} C_VEL
LIN {X 0,Y 118.937,Z 1195.567,A -85,B 0,C 180,E1 31474.646,E2 31474.646} C_VEL
LIN {X 0,Y 186.519,Z 1171.932,A -85,B 0,C 180,E1 31494.925,E2 31494.925} C_VEL
LIN {X 0,Y 209.381,Z 1161.528,A -85,B 0,C 180,E1 31498.39,E2 31498.39} C_VEL
LIN {X 0,Y 225.451,Z 1153.305,A -85,B 0,C 180,E1 31502.559,E2 31502.559} C_VEL
LIN {X 0,Y 152.87,Z 1184.99,A -85,B 0,C 180,E1 31514.304,E2 31514.304} C_VEL
LIN {X 0,Y 92.458,Z 1202.212,A -85,B 0,C 180,E1 31542.413,E2 31542.413} C_VEL
LIN {X 0,Y 74.785,Z 1205.698,A -85,B 0,C 180,E1 31584.164,E2 31584.164} C_VEL
LIN {X 0,Y 81.484,Z 1201.96,A -85,B 0,C 180,E1 31623.297,E2 31623.297} C_VEL
LIN {X 0,Y 127.495,Z 1185.271,A -85,B 0,C 180,E1 31658.749,E2 31658.749} C_VEL
LIN {X 0,Y 194.306,Z 1153.614,A -85,B 0,C 180,E1 31674.243,E2 31674.243} C_VEL
LIN {X 0,Y 261.638,Z 1108.181,A -85,B 0,C 180,E1 31681.338,E2 31681.338} C_VEL
LIN {X 0,Y 285.605,Z 1087.587,A -85,B 0,C 180,E1 31683.121,E2 31683.121} C_VEL
LIN {X 0,Y 220.618,Z 1137.395,A -85,B 0,C 180,E1 31688.888,E2 31688.888} C_VEL
LIN {X 0,Y 153.32,Z 1173.62,A -85,B 0,C 180,E1 31700.035,E2 31700.035} C_VEL
LIN {X 0,Y 95.879,Z 1195.591,A -85,B 0,C 180,E1 31725.521,E2 31725.521} C_VEL
LIN {X 0,Y 75.49,Z 1203.192,A -85,B 0,C 180,E1 31764.252,E2 31764.252} C_VEL
LIN {X 0,Y 77.274,Z 1203.85,A -85,B 0,C 180,E1 31799.399,E2 31799.399} C_VEL
LIN {X 0,Y 114.484,Z 1195.837,A -85,B 0,C 180,E1 31838.035,E2 31838.035} C_VEL
LIN {X 0,Y 183.348,Z 1172.935,A -85,B 0,C 180,E1 31857.171,E2 31857.171} C_VEL
LIN {X 0,Y 225.451,Z 1153.305,A -85,B 0,C 180,E1 31862.559,E2 31862.559} C_VEL
LIN {X 0,Y 193.725,Z 1168.59,A -85,B 0,C 180,E1 31864.076,E2 31864.076} C_VEL
LIN {X 0,Y 120.708,Z 1194.287,A -85,B 0,C 180,E1 31879.54,E2 31879.54} C_VEL
LIN {X 0,Y 72.17,Z 1204.927,A -85,B 0,C 180,E1 31918.291,E2 31918.291} C_VEL
LIN {X 0,Y 66.788,Z 1205.238,A -85,B 0,C 180,E1 31956.5,E2 31956.5} C_VEL
LIN {X 0,Y 88.709,Z 1197.391,A -85,B 0,C 180,E1 32003.361,E2 32003.361} C_VEL
LIN {X 0,Y 150.426,Z 1174.649,A -85,B 0,C 180,E1 32029.345,E2 32029.345} C_VEL
LIN {X 0,Y 219.869,Z 1137.749,A -85,B 0,C 180,E1 32039.635,E2 32039.635} C_VEL
LIN {X 0,Y 262.147,Z 1107.621,A -85,B 0,C 180,E1 32043.21,E2 32043.21} C_VEL
LIN {X 0,Y 195.009,Z 1152.195,A -85,B 0,C 180,E1 32049.543,E2 32049.543} C_VEL
LIN {X 0,Y 127.782,Z 1183.114,A -85,B 0,C 180,E1 32063.138,E2 32063.138} C_VEL
LIN {X 0,Y 75.074,Z 1200.503,A -85,B 0,C 180,E1 32099.689,E2 32099.689} C_VEL
LIN {X 0,Y 66.1,Z 1204.002,A -85,B 0,C 180,E1 32136.606,E2 32136.606} C_VEL
LIN {X 0,Y 84.187,Z 1201.644,A -85,B 0,C 180,E1 32184.179,E2 32184.179} C_VEL
LIN {X 0,Y 149.317,Z 1185.148,A -85,B 0,C 180,E1 32213.785,E2 32213.785} C_VEL
LIN {X 0,Y 204.982,Z 1163.413,A -85,B 0,C 180,E1 32222.762,E2 32222.762} C_VEL
LIN {X 0,Y 193.725,Z 1168.59,A -85,B 0,C 180,E1 32224.076,E2 32224.076} C_VEL
LIN {X 0,Y 178.11,Z 1174.88,A -85,B 0,C 180,E1 32223.059,E2 32223.059} C_VEL
LIN {X 0,Y 162.647,Z 1180.467,A -85,B 0,C 180,E1 32219.642,E2 32219.642} C_VEL
LIN {X 0,Y 90.471,Z 1199.795,A -85,B 0,C 180,E1 32197.242,E2 32197.242} C_VEL
LIN {X 0,Y 59.122,Z 1204.328,A -85,B 0,C 180,E1 32152.651,E2 32152.651} C_VEL
LIN {X 0,Y 59.559,Z 1203.426,A -85,B 0,C 180,E1 32122.707,E2 32122.707} C_VEL
LIN {X 0,Y 91.212,Z 1194.205,A -85,B 0,C 180,E1 32073.794,E2 32073.794} C_VEL
LIN {X 0,Y 158.987,Z 1169.632,A -85,B 0,C 180,E1 32052.169,E2 32052.169} C_VEL
LIN {X 0,Y 228.397,Z 1131.938,A -85,B 0,C 180,E1 32043.855,E2 32043.855} C_VEL
LIN {X 0,Y 235.376,Z 1127.318,A -85,B 0,C 180,E1 32043.112,E2 32043.112} C_VEL
LIN {X 0,Y 165.059,Z 1167.297,A -85,B 0,C 180,E1 32035.402,E2 32035.402} C_VEL
LIN {X 0,Y 96.77,Z 1193.449,A -85,B 0,C 180,E1 32015.981,E2 32015.981} C_VEL
LIN {X 0,Y 60.583,Z 1204.068,A -85,B 0,C 180,E1 31972.031,E2 31972.031} C_VEL
LIN {X 0,Y 58.772,Z 1205.503,A -85,B 0,C 180,E1 31942.566,E2 31942.566} C_VEL
LIN {X 0,Y 85.076,Z 1201.642,A -85,B 0,C 180,E1 31891.639,E2 31891.639} C_VEL
LIN {X 0,Y 156.536,Z 1182.85,A -85,B 0,C 180,E1 31866.727,E2 31866.727} C_VEL
LIN {X 0,Y 181.45,Z 1173.506,A -85,B 0,C 180,E1 31862.348,E2 31862.348} C_VEL
LIN {X 0,Y 162.647,Z 1180.467,A -85,B 0,C 180,E1 31859.642,E2 31859.642} C_VEL
LIN {X 0,Y 129.34,Z 1190.551,A -85,B 0,C 180,E1 31856.762,E2 31856.762} C_VEL
LIN {X 0,Y 64.141,Z 1203.247,A -85,B 0,C 180,E1 31823.588,E2 31823.588} C_VEL
LIN {X 0,Y 49.955,Z 1204.2,A -85,B 0,C 180,E1 31778.756,E2 31778.756} C_VEL
LIN {X 0,Y 61.694,Z 1200.778,A -85,B 0,C 180,E1 31732.11,E2 31732.11} C_VEL
LIN {X 0,Y 122.31,Z 1183.549,A -85,B 0,C 180,E1 31696.116,E2 31696.116} C_VEL
LIN {X 0,Y 196.177,Z 1151.16,A -85,B 0,C 180,E1 31684.469,E2 31684.469} C_VEL
LIN {X 0,Y 209.303,Z 1143.726,A -85,B 0,C 180,E1 31683.122,E2 31683.122} C_VEL
LIN {X 0,Y 139.742,Z 1177.565,A -85,B 0,C 180,E1 31674.194,E2 31674.194} C_VEL
LIN {X 0,Y 76.168,Z 1198.1,A -85,B 0,C 180,E1 31650.272,E2 31650.272} C_VEL
LIN {X 0,Y 50.806,Z 1205.007,A -85,B 0,C 180,E1 31598.558,E2 31598.558} C_VEL
LIN {X 0,Y 58.86,Z 1204.803,A -85,B 0,C 180,E1 31549.874,E2 31549.874} C_VEL
LIN {X 0,Y 116.191,Z 1194.28,A -85,B 0,C 180,E1 31511.75,E2 31511.75} C_VEL
LIN {X 0,Y 162.179,Z 1180.628,A -85,B 0,C 180,E1 31502.627,E2 31502.627} C_VEL
LIN {X 0,Y 129.34,Z 1190.551,A -85,B 0,C 180,E1 31496.762,E2 31496.762} C_VEL
LIN {X 0,Y 95.775,Z 1198.007,A -85,B 0,C 180,E1 31492.213,E2 31492.213} C_VEL
LIN {X 0,Y 50.886,Z 1204.176,A -85,B 0,C 180,E1 31458.198,E2 31458.198} C_VEL
LIN {X 0,Y 43.662,Z 1203.66,A -85,B 0,C 180,E1 31400.029,E2 31400.029} C_VEL
LIN {X 0,Y 83.292,Z 1194.558,A -85,B 0,C 180,E1 31344.486,E2 31344.486} C_VEL
LIN {X 0,Y 156.36,Z 1170.157,A -85,B 0,C 180,E1 31326.303,E2 31326.303} C_VEL
LIN {X 0,Y 182.107,Z 1158.426,A -85,B 0,C 180,E1 31323.157,E2 31323.157} C_VEL
LIN {X 0,Y 107.196,Z 1188.426,A -85,B 0,C 180,E1 31310.908,E2 31310.908} C_VEL
LIN {X 0,Y 50.519,Z 1202.722,A -85,B 0,C 180,E1 31271.615,E2 31271.615} C_VEL
LIN {X 0,Y 42.807,Z 1205.308,A -85,B 0,C 180,E1 31219.768,E2 31219.768} C_VEL
LIN {X 0,Y 80.517,Z 1201.159,A -85,B 0,C 180,E1 31159.615,E2 31159.615} C_VEL
LIN {X 0,Y 138.715,Z 1188.045,A -85,B 0,C 180,E1 31143.071,E2 31143.071} C_VEL
LIN {X 0,Y 95.775,Z 1198.007,A -85,B 0,C 180,E1 31132.213,E2 31132.213} C_VEL
LIN {X 0,Y 62.797,Z 1202.596,A -85,B 0,C 180,E1 31123.272,E2 31123.272} C_VEL
LIN {X 0,Y 33.915,Z 1204.398,A -85,B 0,C 180,E1 31062.957,E2 31062.957} C_VEL
LIN {X 0,Y 41.096,Z 1202.735,A -85,B 0,C 180,E1 31016.429,E2 31016.429} C_VEL
LIN {X 0,Y 100.93,Z 1189.406,A -85,B 0,C 180,E1 30972.472,E2 30972.472} C_VEL
LIN {X 0,Y 152.891,Z 1171.56,A -85,B 0,C 180,E1 30962.9,E2 30962.9} C_VEL
LIN {X 0,Y 77.965,Z 1195.699,A -85,B 0,C 180,E1 30946.469,E2 30946.469} C_VEL
LIN {X 0,Y 39.039,Z 1203.718,A -85,B 0,C 180,E1 30905.599,E2 30905.599} C_VEL
LIN {X 0,Y 34.875,Z 1205.21,A -85,B 0,C 180,E1 30857.406,E2 30857.406} C_VEL
LIN {X 0,Y 78.117,Z 1201.118,A -85,B 0,C 180,E1 30793.854,E2 30793.854} C_VEL
LIN {X 0,Y 118.047,Z 1193.376,A -85,B 0,C 180,E1 30782.545,E2 30782.545} C_VEL
LIN {X 0,Y 62.797,Z 1202.596,A -85,B 0,C 180,E1 30763.272,E2 30763.272} C_VEL
LIN {X 0,Y 32.382,Z 1204.61,A -85,B 0,C 180,E1 30739.711,E2 30739.711} C_VEL
LIN {X 0,Y 27.947,Z 1203.894,A -85,B 0,C 180,E1 30674.304,E2 30674.304} C_VEL
LIN {X 0,Y 77.982,Z 1194.91,A -85,B 0,C 180,E1 30613.584,E2 30613.584} C_VEL
LIN {X 0,Y 126.112,Z 1181.568,A -85,B 0,C 180,E1 30603.517,E2 30603.517} C_VEL
LIN {X 0,Y 55.553,Z 1199.786,A -85,B 0,C 180,E1 30582.748,E2 30582.748} C_VEL
LIN {X 0,Y 27.056,Z 1204.658,A -85,B 0,C 180,E1 30526.227,E2 30526.227} C_VEL
LIN {X 0,Y 43.053,Z 1204.619,A -85,B 0,C 180,E1 30448.228,E2 30448.228} C_VEL
LIN {X 0,Y 92.959,Z 1198.378,A -85,B 0,C 180,E1 30422.144,E2 30422.144} C_VEL
LIN {X 0,Y 32.382,Z 1204.61,A -85,B 0,C 180,E1 30379.711,E2 30379.711} C_VEL
LIN {X 0,Y 21.621,Z 1203.789,A -85,B 0,C 180,E1 30299.818,E2 30299.818} C_VEL
LIN {X 0,Y 83.835,Z 1193.555,A -85,B 0,C 180,E1 30245.948,E2 30245.948} C_VEL
LIN {X 0,Y 97.762,Z 1190.039,A -85,B 0,C 180,E1 30243.245,E2 30243.245} C_VEL
LIN {X 0,Y 39.788,Z 1201.803,A -85,B 0,C 180,E1 30222.23,E2 30222.23} C_VEL
LIN {X 0,Y 19.432,Z 1204.542,A -85,B 0,C 180,E1 30172.896,E2 30172.896} C_VEL
LIN {X 0,Y 39.825,Z 1204.557,A -85,B 0,C 180,E1 30077.729,E2 30077.729} C_VEL
LIN {X 0,Y 71.077,Z 1201.59,A -85,B 0,C 180,E1 30062.542,E2 30062.542} C_VEL
LIN {X 0,Y 18.341,Z 1204.596,A -85,B 0,C 180,E1 29994.495,E2 29994.495} C_VEL
LIN {X 0,Y 21.621,Z 1203.789,A -85,B 0,C 180,E1 29939.818,E2 29939.818} C_VEL
LIN {X 0,Y 45.03,Z 1200.682,A -85,B 0,C 180,E1 29889.485,E2 29889.485} C_VEL
LIN {X 0,Y 65.226,Z 1197.429,A -85,B 0,C 180,E1 29883.125,E2 29883.125} C_VEL
LIN {X 0,Y 12.375,Z 1204.425,A -85,B 0,C 180,E1 29827.658,E2 29827.658} C_VEL
LIN {X 0,Y 38.132,Z 1204.496,A -85,B 0,C 180,E1 29705.848,E2 29705.848} C_VEL
LIN {X 0,Y 44.961,Z 1204.003,A -85,B 0,C 180,E1 29702.602,E2 29702.602} C_VEL
LIN {X 0,Y 13.147,Z 1204.128,A -85,B 0,C 180,E1 29574.896,E2 29574.896} C_VEL
LIN {X 0,Y 45.03,Z 1200.682,A -85,B 0,C 180,E1 29529.485,E2 29529.485} C_VEL
LIN {X 0,Y 22.853,Z 1203.241,A -85,B 0,C 180,E1 29522.132,E2 29522.132} C_VEL
LIN {X 0,Y 9.817,Z 1204.156,A -85,B 0,C 180,E1 29512.3,E2 29512.3} C_VEL
LIN {X 0,Y 7.609,Z 1204.795,A -85,B 0,C 180,E1 29337.943,E2 29337.943} C_VEL
LIN {X 0,Y 22.821,Z 1203.23,A -85,B 0,C 180,E1 29165.259,E2 29165.259} C_VEL
LIN {X 0,Y 9.817,Z 1204.156,A -85,B 0,C 180,E1 29152.3,E2 29152.3} C_VEL
LIN {X 0,Y 8.06,Z 1206.152,A -85,B 0,C 180,E1 29148.318,E2 29148.318} C_VEL
LIN {X 0,Y 8.06,Z 1215,A -85,B 0,C 180,E1 29148.318,E2 29148.318} C_VEL
LIN {X 0,Y 8.06,Z 1215,A -85,B 0,C 180,E1 29148.318,E2 29148.318}

QRS_NEXT_CUT()
PTP {E1 28977.265,E2 28977.265}
PTP {X 0,Y 759.887,A -85,B 0,C 180,E1 28977.265,E2 28977.265,E3 0,E4 0,E5 0,E6 0}
QRS_SPEED_INIT()
LIN {X 0,Y 759.887,Z 1215,A -85,B 0,C 180,E1 28977.265,E2 28977.265,E3 0,E4 0,E5 0,E6 0} C_VEL
LIN {X 0,Y 759.887,Z 329.651,A -85,B 0,C 180,E1 28977.265,E2 28977.265} C_VEL
LIN {X 0,Y 759.887,Z 321.574,A -85,B 0,C 180,E1 28977.265,E2 28977.265} C_VEL
LIN {X 0,Y 759.863,Z 319.574,A -85,B 0,C 180,E1 28977.115,E2 28977.115} C_VEL
LIN {X 0,Y 759.823,Z 319.574,A -85,B 0,C 180,E1 28974.639,E2 28974.639} C_VEL
LIN {X 0,Y 759.821,Z 319.575,A -85,B 0,C 180,E1 28972.362,E2 28972.362} C_VEL
LIN {X 0,Y 759.837,Z 319.575,A -85,B 0,C 180,E1 28969.997,E2 28969.997} C_VEL
LIN {X 0,Y 759.912,Z 319.572,A -85,B 0,C 180,E1 28967.152,E2 28967.152} C_VEL
LIN {X 0,Y 759.834,Z 319.572,A -85,B 0,C 180,E1 28964.416,E2 28964.416} C_VEL
LIN {X 0,Y 759.832,Z 319.574,A -85,B 0,C 180,E1 28962.064,E2 28962.064} C_VEL
LIN {X 0,Y 759.87,Z 319.576,A -85,B 0,C 180,E1 28959.534,E2 28959.534} C_VEL
LIN {X 0,Y 759.864,Z 319.571,A -85,B 0,C 180,E1 28956.502,E2 28956.502} C_VEL
LIN {X 0,Y 759.838,Z 319.573,A -85,B 0,C 180,E1 28953.995,E2 28953.995} C_VEL
LIN {X 0,Y 759.858,Z 319.575,A -85,B 0,C 180,E1 28951.521,E2 28951.521} C_VEL
LIN {X 0,Y 759.914,Z 319.568,A -85,B 0,C 180,E1 28948.597,E2 28948.597} C_VEL
LIN {X 0,Y 759.846,Z 319.572,A -85,B 0,C 180,E1 28945.862,E2 28945.862} C_VEL
LIN {X 0,Y 759.86,Z 319.575,A -85,B 0,C 180,E1 28943.386,E2 28943.386} C_VEL
LIN {X 0,Y 759.914,Z 319.571,A -85,B 0,C 180,E1 28940.541,E2 28940.541} C_VEL
LIN {X 0,Y 759.907,Z 319.724,A -85,B 0,C 180,E1 28938.269,E2 28938.269} C_VEL
LIN {X 0,Y 759.904,Z 341.127,A -85,B 0,C 180,E1 28936.867,E2 28936.867} C_VEL
LIN {X 0,Y 759.919,Z 552.902,A -85,B 0,C 180,E1 28934.32,E2 28934.32} C_VEL
LIN {X 0,Y 759.916,Z 778.42,A -85,B 0,C 180,E1 28931.704,E2 28931.704} C_VEL
LIN {X 0,Y 759.914,Z 820.653,A -85,B 0,C 180,E1 28931.195,E2 28931.195} C_VEL
LIN {X 0,Y 759.905,Z 846.822,A -85,B 0,C 180,E1 28930.74,E2 28930.74} C_VEL
LIN {X 0,Y 759.918,Z 873.65,A -85,B 0,C 180,E1 28930.116,E2 28930.116} C_VEL
LIN {X 0,Y 759.908,Z 896.247,A -85,B 0,C 180,E1 28929.458,E2 28929.458} C_VEL
LIN {X 0,Y 759.918,Z 915.66,A -85,B 0,C 180,E1 28928.806,E2 28928.806} C_VEL
LIN {X 0,Y 759.918,Z 935.317,A -85,B 0,C 180,E1 28928.056,E2 28928.056} C_VEL
LIN {X 0,Y 759.916,Z 959.798,A -85,B 0,C 180,E1 28926.995,E2 28926.995} C_VEL
LIN {X 0,Y 759.916,Z 982.724,A -85,B 0,C 180,E1 28925.839,E2 28925.839} C_VEL
LIN {X 0,Y 759.908,Z 1001.141,A -85,B 0,C 180,E1 28924.808,E2 28924.808} C_VEL
LIN {X 0,Y 759.901,Z 1019.397,A -85,B 0,C 180,E1 28923.683,E2 28923.683} C_VEL
LIN {X 0,Y 759.91,Z 1038.968,A -85,B 0,C 180,E1 28922.355,E2 28922.355} C_VEL
LIN {X 0,Y 759.918,Z 1059.767,A -85,B 0,C 180,E1 28920.772,E2 28920.772} C_VEL
LIN {X 0,Y 759.91,Z 1076.112,A -85,B 0,C 180,E1 28919.392,E2 28919.392} C_VEL
LIN {X 0,Y 759.915,Z 1093.679,A -85,B 0,C 180,E1 28917.761,E2 28917.761} C_VEL
LIN {X 0,Y 759.898,Z 1110.594,A -85,B 0,C 180,E1 28915.986,E2 28915.986} C_VEL
LIN {X 0,Y 759.907,Z 1123.447,A -85,B 0,C 180,E1 28914.486,E2 28914.486} C_VEL
LIN {X 0,Y 759.893,Z 1134.935,A -85,B 0,C 180,E1 28913.004,E2 28913.004} C_VEL
LIN {X 0,Y 759.912,Z 1145.719,A -85,B 0,C 180,E1 28911.456,E2 28911.456} C_VEL
LIN {X 0,Y 759.914,Z 1157.63,A -85,B 0,C 180,E1 28909.524,E2 28909.524} C_VEL
LIN {X 0,Y 759.909,Z 1167.862,A -85,B 0,C 180,E1 28907.536,E2 28907.536} C_VEL
LIN {X 0,Y 759.908,Z 1175.846,A -85,B 0,C 180,E1 28905.727,E2 28905.727} C_VEL
LIN {X 0,Y 759.909,Z 1183.258,A -85,B 0,C 180,E1 28903.622,E2 28903.622} C_VEL
LIN {X 0,Y 759.917,Z 1188.604,A -85,B 0,C 180,E1 28901.613,E2 28901.613} C_VEL
LIN {X 0,Y 759.912,Z 1192.323,A -85,B 0,C 180,E1 28899.619,E2 28899.619} C_VEL
LIN {X 0,Y 759.911,Z 1194.533,A -85,B 0,C 180,E1 28897.484,E2 28897.484} C_VEL
LIN {X 0,Y 759.892,Z 1194.874,A -85,B 0,C 180,E1 28895.512,E2 28895.512} C_VEL
LIN {X 0,Y 759.907,Z 1193.91,A -85,B 0,C 180,E1 28893.621,E2 28893.621} C_VEL
LIN {X 0,Y 759.908,Z 1191.062,A -85,B 0,C 180,E1 28891.508,E2 28891.508} C_VEL
LIN {X 0,Y 759.915,Z 1186.603,A -85,B 0,C 180,E1 28889.472,E2 28889.472} C_VEL
LIN {X 0,Y 759.914,Z 1180.736,A -85,B 0,C 180,E1 28887.511,E2 28887.511} C_VEL
LIN {X 0,Y 759.889,Z 1172.595,A -85,B 0,C 180,E1 28885.396,E2 28885.396} C_VEL
LIN {X 0,Y 759.91,Z 1163.165,A -85,B 0,C 180,E1 28883.426,E2 28883.426} C_VEL
LIN {X 0,Y 759.914,Z 1154.301,A -85,B 0,C 180,E1 28881.83,E2 28881.83} C_VEL
LIN {X 0,Y 759.902,Z 1144.345,A -85,B 0,C 180,E1 28880.248,E2 28880.248} C_VEL
LIN {X 0,Y 759.911,Z 1133.929,A -85,B 0,C 180,E1 28878.77,E2 28878.77} C_VEL
LIN {X 0,Y 759.898,Z 1121.238,A -85,B 0,C 180,E1 28877.151,E2 28877.151} C_VEL
LIN {X 0,Y 759.891,Z 1104.021,A -85,B 0,C 180,E1 28875.21,E2 28875.21} C_VEL
LIN {X 0,Y 759.904,Z 1089.214,A -85,B 0,C 180,E1 28873.724,E2 28873.724} C_VEL
LIN {X 0,Y 759.912,Z 1073.6,A -85,B 0,C 180,E1 28872.296,E2 28872.296} C_VEL
LIN {X 0,Y 759.907,Z 1052.915,A -85,B 0,C 180,E1 28870.595,E2 28870.595} C_VEL
LIN {X 0,Y 759.903,Z 1034.314,A -85,B 0,C 180,E1 28869.23,E2 28869.23} C_VEL
LIN {X 0,Y 759.901,Z 1016.123,A -85,B 0,C 180,E1 28868.016,E2 28868.016} C_VEL
LIN {X 0,Y 759.905,Z 993.032,A -85,B 0,C 180,E1 28866.627,E2 28866.627} C_VEL
LIN {X 0,Y 759.918,Z 971.117,A -85,B 0,C 180,E1 28865.473,E2 28865.473} C_VEL
LIN {X 0,Y 759.912,Z 951.775,A -85,B 0,C 180,E1 28864.557,E2 28864.557} C_VEL
LIN {X 0,Y 759.918,Z 933.002,A -85,B 0,C 180,E1 28863.762,E2 28863.762} C_VEL
LIN {X 0,Y 759.919,Z 914.01,A -85,B 0,C 180,E1 28863.045,E2 28863.045} C_VEL
LIN {X 0,Y 759.908,Z 896.029,A -85,B 0,C 180,E1 28862.445,E2 28862.445} C_VEL
LIN {X 0,Y 759.908,Z 873.537,A -85,B 0,C 180,E1 28861.79,E2 28861.79} C_VEL
LIN {X 0,Y 759.916,Z 845.576,A -85,B 0,C 180,E1 28861.145,E2 28861.145} C_VEL
LIN {X 0,Y 759.908,Z 818.488,A -85,B 0,C 180,E1 28860.683,E2 28860.683} C_VEL
LIN {X 0,Y 759.91,Z 567.957,A -85,B 0,C 180,E1 28857.767,E2 28857.767} C_VEL
LIN {X 0,Y 759.909,Z 354.793,A -85,B 0,C 180,E1 28855.211,E2 28855.211} C_VEL
LIN {X 0,Y 759.91,Z 340.626,A -85,B 0,C 180,E1 28855.026,E2 28855.026} C_VEL
LIN {X 0,Y 759.896,Z 319.574,A -85,B 0,C 180,E1 28853.619,E2 28853.619} C_VEL
LIN {X 0,Y 759.896,Z 319.575,A -85,B 0,C 180,E1 28850.807,E2 28850.807} C_VEL
LIN {X 0,Y 759.909,Z 319.564,A -85,B 0,C 180,E1 28847.912,E2 28847.912} C_VEL
LIN {X 0,Y 759.906,Z 319.576,A -85,B 0,C 180,E1 28844.829,E2 28844.829} C_VEL
LIN {X 0,Y 759.888,Z 319.567,A -85,B 0,C 180,E1 28841.948,E2 28841.948} C_VEL
LIN {X 0,Y 759.906,Z 319.573,A -85,B 0,C 180,E1 28839.07,E2 28839.07} C_VEL
LIN {X 0,Y 759.872,Z 319.572,A -85,B 0,C 180,E1 28836.309,E2 28836.309} C_VEL
LIN {X 0,Y 759.902,Z 319.566,A -85,B 0,C 180,E1 28833.549,E2 28833.549} C_VEL
LIN {X 0,Y 759.894,Z 319.576,A -85,B 0,C 180,E1 28830.525,E2 28830.525} C_VEL
LIN {X 0,Y 759.863,Z 319.57,A -85,B 0,C 180,E1 28827.839,E2 28827.839} C_VEL
LIN {X 0,Y 759.912,Z 319.567,A -85,B 0,C 180,E1 28825.068,E2 28825.068} C_VEL
LIN {X 0,Y 759.87,Z 319.574,A -85,B 0,C 180,E1 28822.189,E2 28822.189} C_VEL
LIN {X 0,Y 759.857,Z 319.569,A -85,B 0,C 180,E1 28819.581,E2 28819.581} C_VEL
LIN {X 0,Y 759.914,Z 319.57,A -85,B 0,C 180,E1 28816.827,E2 28816.827} C_VEL
LIN {X 0,Y 759.861,Z 319.573,A -85,B 0,C 180,E1 28814.012,E2 28814.012} C_VEL
LIN {X 0,Y 759.845,Z 319.572,A -85,B 0,C 180,E1 28811.538,E2 28811.538} C_VEL
LIN {X 0,Y 759.888,Z 319.569,A -85,B 0,C 180,E1 28808.932,E2 28808.932} C_VEL
LIN {X 0,Y 759.865,Z 319.575,A -85,B 0,C 180,E1 28805.967,E2 28805.967} C_VEL
LIN {X 0,Y 759.835,Z 319.574,A -85,B 0,C 180,E1 28803.546,E2 28803.546} C_VEL
LIN {X 0,Y 759.84,Z 319.572,A -85,B 0,C 180,E1 28801.131,E2 28801.131} C_VEL
LIN {X 0,Y 759.918,Z 319.574,A -85,B 0,C 180,E1 28798.341,E2 28798.341} C_VEL
LIN {X 0,Y 759.835,Z 319.575,A -85,B 0,C 180,E1 28795.547,E2 28795.547} C_VEL
LIN {X 0,Y 759.822,Z 319.575,A -85,B 0,C 180,E1 28793.198,E2 28793.198} C_VEL
LIN {X 0,Y 759.83,Z 319.574,A -85,B 0,C 180,E1 28790.838,E2 28790.838} C_VEL
LIN {X 0,Y 759.919,Z 319.576,A -85,B 0,C 180,E1 28788.078,E2 28788.078} C_VEL
LIN {X 0,Y 759.824,Z 319.576,A -85,B 0,C 180,E1 28785.365,E2 28785.365} C_VEL
LIN {X 0,Y 759.809,Z 319.577,A -85,B 0,C 180,E1 28783.078,E2 28783.078} C_VEL
LIN {X 0,Y 759.806,Z 319.576,A -85,B 0,C 180,E1 28780.872,E2 28780.872} C_VEL
LIN {X 0,Y 759.811,Z 319.577,A -85,B 0,C 180,E1 28778.622,E2 28778.622} C_VEL
LIN {X 0,Y 759.892,Z 319.578,A -85,B 0,C 180,E1 28775.948,E2 28775.948} C_VEL
LIN {X 0,Y 759.82,Z 319.577,A -85,B 0,C 180,E1 28773.152,E2 28773.152} C_VEL
LIN {X 0,Y 759.807,Z 319.577,A -85,B 0,C 180,E1 28770.862,E2 28770.862} C_VEL
LIN {X 0,Y 759.809,Z 319.576,A -85,B 0,C 180,E1 28768.656,E2 28768.656} C_VEL
LIN {X 0,Y 759.816,Z 319.577,A -85,B 0,C 180,E1 28766.447,E2 28766.447} C_VEL
LIN {X 0,Y 759.873,Z 319.577,A -85,B 0,C 180,E1 28763.878,E2 28763.878} C_VEL
LIN {X 0,Y 759.841,Z 319.575,A -85,B 0,C 180,E1 28760.926,E2 28760.926} C_VEL
LIN {X 0,Y 759.824,Z 319.575,A -85,B 0,C 180,E1 28758.553,E2 28758.553} C_VEL
LIN {X 0,Y 759.828,Z 319.576,A -85,B 0,C 180,E1 28756.257,E2 28756.257} C_VEL
LIN {X 0,Y 759.889,Z 319.578,A -85,B 0,C 180,E1 28753.638,E2 28753.638} C_VEL
LIN {X 0,Y 759.875,Z 319.624,A -85,B 0,C 180,E1 28752.944,E2 28752.944} C_VEL
LIN {X 0,Y 759.894,Z 350.883,A -85,B 0,C 180,E1 28750.916,E2 28750.916} C_VEL
LIN {X 0,Y 759.915,Z 561.445,A -85,B 0,C 180,E1 28748.382,E2 28748.382} C_VEL
LIN {X 0,Y 759.92,Z 788.585,A -85,B 0,C 180,E1 28745.747,E2 28745.747} C_VEL
LIN {X 0,Y 759.911,Z 831.13,A -85,B 0,C 180,E1 28745.233,E2 28745.233} C_VEL
LIN {X 0,Y 759.91,Z 856.582,A -85,B 0,C 180,E1 28744.789,E2 28744.789} C_VEL
LIN {X 0,Y 759.913,Z 883.584,A -85,B 0,C 180,E1 28744.163,E2 28744.163} C_VEL
LIN {X 0,Y 759.907,Z 907.507,A -85,B 0,C 180,E1 28743.465,E2 28743.465} C_VEL
LIN {X 0,Y 759.918,Z 932.857,A -85,B 0,C 180,E1 28742.597,E2 28742.597} C_VEL
LIN {X 0,Y 759.917,Z 957.684,A -85,B 0,C 180,E1 28741.579,E2 28741.579} C_VEL
LIN {X 0,Y 759.913,Z 976.725,A -85,B 0,C 180,E1 28740.699,E2 28740.699} C_VEL
LIN {X 0,Y 759.913,Z 995.409,A -85,B 0,C 180,E1 28739.739,E2 28739.739} C_VEL
LIN {X 0,Y 759.909,Z 1013.692,A -85,B 0,C 180,E1 28738.703,E2 28738.703} C_VEL
LIN {X 0,Y 759.913,Z 1035.188,A -85,B 0,C 180,E1 28737.356,E2 28737.356} C_VEL
LIN {X 0,Y 759.91,Z 1056.55,A -85,B 0,C 180,E1 28735.84,E2 28735.84} C_VEL
LIN {X 0,Y 759.914,Z 1073.305,A -85,B 0,C 180,E1 28734.528,E2 28734.528} C_VEL
LIN {X 0,Y 759.897,Z 1092.039,A -85,B 0,C 180,E1 28732.915,E2 28732.915} C_VEL
LIN {X 0,Y 759.895,Z 1109.488,A -85,B 0,C 180,E1 28731.214,E2 28731.214} C_VEL
LIN {X 0,Y 759.905,Z 1122.952,A -85,B 0,C 180,E1 28729.765,E2 28729.765} C_VEL
LIN {X 0,Y 759.897,Z 1135.726,A -85,B 0,C 180,E1 28728.25,E2 28728.25} C_VEL
LIN {X 0,Y 759.909,Z 1150.027,A -85,B 0,C 180,E1 28726.355,E2 28726.355} C_VEL
LIN {X 0,Y 759.909,Z 1162.191,A -85,B 0,C 180,E1 28724.478,E2 28724.478} C_VEL
LIN {X 0,Y 759.91,Z 1171.056,A -85,B 0,C 180,E1 28722.926,E2 28722.926} C_VEL
LIN {X 0,Y 759.91,Z 1178.782,A -85,B 0,C 180,E1 28721.383,E2 28721.383} C_VEL
LIN {X 0,Y 759.905,Z 1186.428,A -85,B 0,C 180,E1 28719.62,E2 28719.62} C_VEL
LIN {X 0,Y 759.908,Z 1193.593,A -85,B 0,C 180,E1 28717.561,E2 28717.561} C_VEL
LIN {X 0,Y 759.91,Z 1199.107,A -85,B 0,C 180,E1 28715.436,E2 28715.436} C_VEL
LIN {X 0,Y 759.916,Z 1202.585,A -85,B 0,C 180,E1 28713.47,E2 28713.47} C_VEL
LIN {X 0,Y 759.914,Z 1204.58,A -85,B 0,C 180,E1 28711.433,E2 28711.433} C_VEL
LIN {X 0,Y 759.889,Z 1204.849,A -85,B 0,C 180,E1 28709.473,E2 28709.473} C_VEL
LIN {X 0,Y 759.907,Z 1203.907,A -85,B 0,C 180,E1 28707.663,E2 28707.663} C_VEL
LIN {X 0,Y 759.908,Z 1201.054,A -85,B 0,C 180,E1 28705.548,E2 28705.548} C_VEL
LIN {X 0,Y 759.914,Z 1196.567,A -85,B 0,C 180,E1 28703.503,E2 28703.503} C_VEL
LIN {X 0,Y 759.913,Z 1190.63,A -85,B 0,C 180,E1 28701.526,E2 28701.526} C_VEL
LIN {X 0,Y 759.896,Z 1182.681,A -85,B 0,C 180,E1 28699.462,E2 28699.462} C_VEL
LIN {X 0,Y 759.905,Z 1173.111,A -85,B 0,C 180,E1 28697.461,E2 28697.461} C_VEL
LIN {X 0,Y 759.91,Z 1164.056,A -85,B 0,C 180,E1 28695.834,E2 28695.834} C_VEL
LIN {X 0,Y 759.894,Z 1154.212,A -85,B 0,C 180,E1 28694.273,E2 28694.273} C_VEL
LIN {X 0,Y 759.904,Z 1143.666,A -85,B 0,C 180,E1 28692.78,E2 28692.78} C_VEL
LIN {X 0,Y 759.896,Z 1130.456,A -85,B 0,C 180,E1 28691.1,E2 28691.1} C_VEL
LIN {X 0,Y 759.898,Z 1113.393,A -85,B 0,C 180,E1 28689.191,E2 28689.191} C_VEL
LIN {X 0,Y 759.898,Z 1098.827,A -85,B 0,C 180,E1 28687.732,E2 28687.732} C_VEL
LIN {X 0,Y 759.911,Z 1082.652,A -85,B 0,C 180,E1 28686.258,E2 28686.258} C_VEL
LIN {X 0,Y 759.91,Z 1061.272,A -85,B 0,C 180,E1 28684.516,E2 28684.516} C_VEL
LIN {X 0,Y 759.91,Z 1044.046,A -85,B 0,C 180,E1 28683.257,E2 28683.257} C_VEL
LIN {X 0,Y 759.914,Z 1026.239,A -85,B 0,C 180,E1 28682.069,E2 28682.069} C_VEL
LIN {X 0,Y 759.905,Z 1003.449,A -85,B 0,C 180,E1 28680.694,E2 28680.694} C_VEL
LIN {X 0,Y 759.916,Z 981.266,A -85,B 0,C 180,E1 28679.525,E2 28679.525} C_VEL
LIN {X 0,Y 759.912,Z 961.675,A -85,B 0,C 180,E1 28678.598,E2 28678.598} C_VEL
LIN {X 0,Y 759.918,Z 942.461,A -85,B 0,C 180,E1 28677.785,E2 28677.785} C_VEL
LIN {X 0,Y 759.919,Z 923.844,A -85,B 0,C 180,E1 28677.084,E2 28677.084} C_VEL
LIN {X 0,Y 759.909,Z 905.502,A -85,B 0,C 180,E1 28676.473,E2 28676.473} C_VEL
LIN {X 0,Y 759.913,Z 882.821,A -85,B 0,C 180,E1 28675.818,E2 28675.818} C_VEL
LIN {X 0,Y 759.911,Z 855.67,A -85,B 0,C 180,E1 28675.191,E2 28675.191} C_VEL
LIN {X 0,Y 759.91,Z 829.082,A -85,B 0,C 180,E1 28674.737,E2 28674.737} C_VEL
LIN {X 0,Y 759.915,Z 733.181,A -85,B 0,C 180,E1 28673.619,E2 28673.619} C_VEL
LIN {X 0,Y 759.914,Z 509.74,A -85,B 0,C 180,E1 28671.004,E2 28671.004} C_VEL
LIN {X 0,Y 759.896,Z 350.368,A -85,B 0,C 180,E1 28669.06,E2 28669.06} C_VEL
LIN {X 0,Y 759.879,Z 319.577,A -85,B 0,C 180,E1 28667.032,E2 28667.032} C_VEL
LIN {X 0,Y 759.855,Z 319.577,A -85,B 0,C 180,E1 28664.072,E2 28664.072} C_VEL
LIN {X 0,Y 759.826,Z 319.575,A -85,B 0,C 180,E1 28661.631,E2 28661.631} C_VEL
LIN {X 0,Y 759.827,Z 319.575,A -85,B 0,C 180,E1 28659.308,E2 28659.308} C_VEL
LIN {X 0,Y 759.899,Z 319.573,A -85,B 0,C 180,E1 28656.618,E2 28656.618} C_VEL
LIN {X 0,Y 759.834,Z 319.576,A -85,B 0,C 180,E1 28653.731,E2 28653.731} C_VEL
LIN {X 0,Y 759.816,Z 319.575,A -85,B 0,C 180,E1 28651.408,E2 28651.408} C_VEL
LIN {X 0,Y 759.812,Z 319.576,A -85,B 0,C 180,E1 28649.224,E2 28649.224} C_VEL
LIN {X 0,Y 759.815,Z 319.575,A -85,B 0,C 180,E1 28647.001,E2 28647.001} C_VEL
LIN {X 0,Y 759.859,Z 319.575,A -85,B 0,C 180,E1 28644.488,E2 28644.488} C_VEL
LIN {X 0,Y 759.829,Z 319.576,A -85,B 0,C 180,E1 28641.511,E2 28641.511} C_VEL
LIN {X 0,Y 759.807,Z 319.577,A -85,B 0,C 180,E1 28639.208,E2 28639.208} C_VEL
LIN {X 0,Y 759.8,Z 319.576,A -85,B 0,C 180,E1 28636.987,E2 28636.987} C_VEL
LIN {X 0,Y 759.801,Z 319.577,A -85,B 0,C 180,E1 28634.792,E2 28634.792} C_VEL
LIN {X 0,Y 759.82,Z 319.577,A -85,B 0,C 180,E1 28632.464,E2 28632.464} C_VEL
LIN {X 0,Y 759.886,Z 319.577,A -85,B 0,C 180,E1 28629.62,E2 28629.62} C_VEL
LIN {X 0,Y 759.818,Z 319.576,A -85,B 0,C 180,E1 28627.03,E2 28627.03} C_VEL
LIN {X 0,Y 759.81,Z 319.576,A -85,B 0,C 180,E1 28624.756,E2 28624.756} C_VEL
LIN {X 0,Y 759.812,Z 319.576,A -85,B 0,C 180,E1 28622.564,E2 28622.564} C_VEL
LIN {X 0,Y 759.828,Z 319.575,A -85,B 0,C 180,E1 28620.226,E2 28620.226} C_VEL
LIN {X 0,Y 759.905,Z 319.573,A -85,B 0,C 180,E1 28617.36,E2 28617.36} C_VEL
LIN {X 0,Y 759.863,Z 319.574,A -85,B 0,C 180,E1 28617.115,E2 28617.115} C_VEL
LIN {X 0,Y 758.82,Z 319.702,A -85,B 0,C 180,E1 28616.534,E2 28616.534} C_VEL
LIN {X 0,Y 752.406,Z 320.499,A -85,B 0,C 180,E1 28614.906,E2 28614.906} C_VEL
LIN {X 0,Y 751.88,Z 320.562,A -85,B 0,C 180,E1 28614.484,E2 28614.484} C_VEL
LIN {X 0,Y 751.891,Z 320.565,A -85,B 0,C 180,E1 28612.127,E2 28612.127} C_VEL
LIN {X 0,Y 751.98,Z 320.563,A -85,B 0,C 180,E1 28609.349,E2 28609.349} C_VEL
LIN {X 0,Y 751.898,Z 320.562,A -85,B 0,C 180,E1 28606.543,E2 28606.543} C_VEL
LIN {X 0,Y 751.891,Z 320.56,A -85,B 0,C 180,E1 28604.18,E2 28604.18} C_VEL
LIN {X 0,Y 751.915,Z 320.565,A -85,B 0,C 180,E1 28601.704,E2 28601.704} C_VEL
LIN {X 0,Y 751.945,Z 320.56,A -85,B 0,C 180,E1 28598.714,E2 28598.714} C_VEL
LIN {X 0,Y 751.9,Z 320.561,A -85,B 0,C 180,E1 28596.155,E2 28596.155} C_VEL
LIN {X 0,Y 751.909,Z 320.564,A -85,B 0,C 180,E1 28593.671,E2 28593.671} C_VEL
LIN {X 0,Y 751.977,Z 320.562,A -85,B 0,C 180,E1 28590.877,E2 28590.877} C_VEL
LIN {X 0,Y 751.916,Z 320.56,A -85,B 0,C 180,E1 28588.134,E2 28588.134} C_VEL
LIN {X 0,Y 751.91,Z 320.564,A -85,B 0,C 180,E1 28585.586,E2 28585.586} C_VEL
LIN {X 0,Y 751.977,Z 320.566,A -85,B 0,C 180,E1 28582.866,E2 28582.866} C_VEL
LIN {X 0,Y 751.927,Z 320.562,A -85,B 0,C 180,E1 28579.99,E2 28579.99} C_VEL
LIN {X 0,Y 751.98,Z 320.592,A -85,B 0,C 180,E1 28578.762,E2 28578.762} C_VEL
LIN {X 0,Y 753.28,Z 324.316,A -85,B 0,C 180,E1 28578.418,E2 28578.418} C_VEL
LIN {X 0,Y 753.325,Z 341.307,A -85,B 0,C 180,E1 28577.3,E2 28577.3} C_VEL
LIN {X 0,Y 753.844,Z 344.375,A -85,B 0,C 180,E1 28577.227,E2 28577.227} C_VEL
LIN {X 0,Y 753.63,Z 557.312,A -85,B 0,C 180,E1 28574.647,E2 28574.647} C_VEL
LIN {X 0,Y 753.408,Z 784.185,A -85,B 0,C 180,E1 28571.994,E2 28571.994} C_VEL
LIN {X 0,Y 753.353,Z 822.782,A -85,B 0,C 180,E1 28571.517,E2 28571.517} C_VEL
LIN {X 0,Y 753.267,Z 849.043,A -85,B 0,C 180,E1 28571.044,E2 28571.044} C_VEL
LIN {X 0,Y 753.187,Z 875.589,A -85,B 0,C 180,E1 28570.412,E2 28570.412} C_VEL
LIN {X 0,Y 753.088,Z 902.188,A -85,B 0,C 180,E1 28569.617,E2 28569.617} C_VEL
LIN {X 0,Y 752.953,Z 927.9,A -85,B 0,C 180,E1 28568.689,E2 28568.689} C_VEL
LIN {X 0,Y 752.857,Z 948.684,A -85,B 0,C 180,E1 28567.82,E2 28567.82} C_VEL
LIN {X 0,Y 752.754,Z 968.214,A -85,B 0,C 180,E1 28566.904,E2 28566.904} C_VEL
LIN {X 0,Y 752.664,Z 987.331,A -85,B 0,C 180,E1 28565.905,E2 28565.905} C_VEL
LIN {X 0,Y 752.554,Z 1008.855,A -85,B 0,C 180,E1 28564.656,E2 28564.656} C_VEL
LIN {X 0,Y 752.427,Z 1031.088,A -85,B 0,C 180,E1 28563.195,E2 28563.195} C_VEL
LIN {X 0,Y 752.342,Z 1048.389,A -85,B 0,C 180,E1 28561.934,E2 28561.934} C_VEL
LIN {X 0,Y 752.262,Z 1066.166,A -85,B 0,C 180,E1 28560.513,E2 28560.513} C_VEL
LIN {X 0,Y 752.174,Z 1085.975,A -85,B 0,C 180,E1 28558.74,E2 28558.74} C_VEL
LIN {X 0,Y 752.112,Z 1100.439,A -85,B 0,C 180,E1 28557.3,E2 28557.3} C_VEL
LIN {X 0,Y 752.07,Z 1114.41,A -85,B 0,C 180,E1 28555.769,E2 28555.769} C_VEL
LIN {X 0,Y 752.024,Z 1129.568,A -85,B 0,C 180,E1 28553.923,E2 28553.923} C_VEL
LIN {X 0,Y 751.957,Z 1143.092,A -85,B 0,C 180,E1 28552.022,E2 28552.022} C_VEL
LIN {X 0,Y 751.959,Z 1152.902,A -85,B 0,C 180,E1 28550.469,E2 28550.469} C_VEL
LIN {X 0,Y 751.924,Z 1161.519,A -85,B 0,C 180,E1 28548.933,E2 28548.933} C_VEL
LIN {X 0,Y 751.93,Z 1169.389,A -85,B 0,C 180,E1 28547.329,E2 28547.329} C_VEL
LIN {X 0,Y 751.92,Z 1177.095,A -85,B 0,C 180,E1 28545.502,E2 28545.502} C_VEL
LIN {X 0,Y 751.913,Z 1183.771,A -85,B 0,C 180,E1 28543.535,E2 28543.535} C_VEL
LIN {X 0,Y 751.911,Z 1189.156,A -85,B 0,C 180,E1 28541.428,E2 28541.428} C_VEL
LIN {X 0,Y 751.915,Z 1192.65,A -85,B 0,C 180,E1 28539.413,E2 28539.413} C_VEL
LIN {X 0,Y 751.913,Z 1194.578,A -85,B 0,C 180,E1 28537.411,E2 28537.411} C_VEL
LIN {X 0,Y 751.896,Z 1194.848,A -85,B 0,C 180,E1 28535.417,E2 28535.417} C_VEL
LIN {X 0,Y 751.906,Z 1193.897,A -85,B 0,C 180,E1 28533.583,E2 28533.583} C_VEL
LIN {X 0,Y 751.907,Z 1191.041,A -85,B 0,C 180,E1 28531.447,E2 28531.447} C_VEL
LIN {X 0,Y 751.912,Z 1186.571,A -85,B 0,C 180,E1 28529.39,E2 28529.39} C_VEL
LIN {X 0,Y 751.921,Z 1180.693,A -85,B 0,C 180,E1 28527.408,E2 28527.408} C_VEL
LIN {X 0,Y 751.905,Z 1172.546,A -85,B 0,C 180,E1 28525.27,E2 28525.27} C_VEL
LIN {X 0,Y 751.943,Z 1163.105,A -85,B 0,C 180,E1 28523.28,E2 28523.28} C_VEL
LIN {X 0,Y 751.951,Z 1153.963,A -85,B 0,C 180,E1 28521.62,E2 28521.62} C_VEL
LIN {X 0,Y 751.965,Z 1144.132,A -85,B 0,C 180,E1 28520.046,E2 28520.046} C_VEL
LIN {X 0,Y 751.997,Z 1133.285,A -85,B 0,C 180,E1 28518.495,E2 28518.495} C_VEL
LIN {X 0,Y 752.059,Z 1118.639,A -85,B 0,C 180,E1 28516.624,E2 28516.624} C_VEL
LIN {X 0,Y 752.092,Z 1102.415,A -85,B 0,C 180,E1 28514.817,E2 28514.817} C_VEL
LIN {X 0,Y 752.173,Z 1087.462,A -85,B 0,C 180,E1 28513.313,E2 28513.313} C_VEL
LIN {X 0,Y 752.251,Z 1069.017,A -85,B 0,C 180,E1 28511.632,E2 28511.632} C_VEL
LIN {X 0,Y 752.332,Z 1049.598,A -85,B 0,C 180,E1 28510.068,E2 28510.068} C_VEL
LIN {X 0,Y 752.407,Z 1031.857,A -85,B 0,C 180,E1 28508.769,E2 28508.769} C_VEL
LIN {X 0,Y 752.564,Z 1009.559,A -85,B 0,C 180,E1 28507.296,E2 28507.296} C_VEL
LIN {X 0,Y 752.663,Z 987.493,A -85,B 0,C 180,E1 28506.014,E2 28506.014} C_VEL
LIN {X 0,Y 752.759,Z 968.361,A -85,B 0,C 180,E1 28505.014,E2 28505.014} C_VEL
LIN {X 0,Y 752.853,Z 949.636,A -85,B 0,C 180,E1 28504.133,E2 28504.133} C_VEL
LIN {X 0,Y 752.949,Z 929.539,A -85,B 0,C 180,E1 28503.288,E2 28503.288} C_VEL
LIN {X 0,Y 753.065,Z 904.614,A -85,B 0,C 180,E1 28502.371,E2 28502.371} C_VEL
LIN {X 0,Y 753.176,Z 876.216,A -85,B 0,C 180,E1 28501.514,E2 28501.514} C_VEL
LIN {X 0,Y 753.277,Z 850.154,A -85,B 0,C 180,E1 28500.89,E2 28500.89} C_VEL
LIN {X 0,Y 753.347,Z 823.693,A -85,B 0,C 180,E1 28500.406,E2 28500.406} C_VEL
LIN {X 0,Y 753.402,Z 786.84,A -85,B 0,C 180,E1 28499.946,E2 28499.946} C_VEL
LIN {X 0,Y 753.621,Z 559.551,A -85,B 0,C 180,E1 28497.29,E2 28497.29} C_VEL
LIN {X 0,Y 753.851,Z 345.929,A -85,B 0,C 180,E1 28494.703,E2 28494.703} C_VEL
LIN {X 0,Y 753.619,Z 342.368,A -85,B 0,C 180,E1 28494.643,E2 28494.643} C_VEL
LIN {X 0,Y 753.218,Z 340.819,A -85,B 0,C 180,E1 28494.596,E2 28494.596} C_VEL
LIN {X 0,Y 753.094,Z 323.787,A -85,B 0,C 180,E1 28493.443,E2 28493.443} C_VEL
LIN {X 0,Y 751.974,Z 320.566,A -85,B 0,C 180,E1 28493.129,E2 28493.129} C_VEL
LIN {X 0,Y 751.95,Z 320.558,A -85,B 0,C 180,E1 28490.227,E2 28490.227} C_VEL
LIN {X 0,Y 751.96,Z 320.559,A -85,B 0,C 180,E1 28487.405,E2 28487.405} C_VEL
LIN {X 0,Y 751.947,Z 320.563,A -85,B 0,C 180,E1 28484.596,E2 28484.596} C_VEL
LIN {X 0,Y 751.967,Z 320.554,A -85,B 0,C 180,E1 28481.759,E2 28481.759} C_VEL
LIN {X 0,Y 751.961,Z 320.565,A -85,B 0,C 180,E1 28478.68,E2 28478.68} C_VEL
LIN {X 0,Y 751.938,Z 320.557,A -85,B 0,C 180,E1 28475.904,E2 28475.904} C_VEL
LIN {X 0,Y 751.968,Z 320.56,A -85,B 0,C 180,E1 28473.102,E2 28473.102} C_VEL
LIN {X 0,Y 751.937,Z 320.563,A -85,B 0,C 180,E1 28470.345,E2 28470.345} C_VEL
LIN {X 0,Y 751.934,Z 320.557,A -85,B 0,C 180,E1 28467.651,E2 28467.651} C_VEL
LIN {X 0,Y 751.974,Z 320.562,A -85,B 0,C 180,E1 28464.747,E2 28464.747} C_VEL
LIN {X 0,Y 751.921,Z 320.561,A -85,B 0,C 180,E1 28462.024,E2 28462.024} C_VEL
LIN {X 0,Y 751.93,Z 320.556,A -85,B 0,C 180,E1 28459.417,E2 28459.417} C_VEL
LIN {X 0,Y 751.969,Z 320.566,A -85,B 0,C 180,E1 28456.453,E2 28456.453} C_VEL
LIN {X 0,Y 751.909,Z 320.559,A -85,B 0,C 180,E1 28453.771,E2 28453.771} C_VEL
LIN {X 0,Y 751.919,Z 320.559,A -85,B 0,C 180,E1 28451.273,E2 28451.273} C_VEL
LIN {X 0,Y 751.97,Z 320.566,A -85,B 0,C 180,E1 28448.334,E2 28448.334} C_VEL
LIN {X 0,Y 751.901,Z 320.563,A -85,B 0,C 180,E1 28445.647,E2 28445.647} C_VEL
LIN {X 0,Y 751.901,Z 320.562,A -85,B 0,C 180,E1 28443.202,E2 28443.202} C_VEL
LIN {X 0,Y 751.979,Z 320.562,A -85,B 0,C 180,E1 28440.381,E2 28440.381} C_VEL
LIN {X 0,Y 751.896,Z 320.564,A -85,B 0,C 180,E1 28437.561,E2 28437.561} C_VEL
LIN {X 0,Y 751.887,Z 320.563,A -85,B 0,C 180,E1 28435.194,E2 28435.194} C_VEL
LIN {X 0,Y 751.908,Z 320.563,A -85,B 0,C 180,E1 28432.742,E2 28432.742} C_VEL
LIN {X 0,Y 751.923,Z 320.566,A -85,B 0,C 180,E1 28429.736,E2 28429.736} C_VEL
LIN {X 0,Y 751.878,Z 320.563,A -85,B 0,C 180,E1 28427.246,E2 28427.246} C_VEL
LIN {X 0,Y 751.873,Z 320.564,A -85,B 0,C 180,E1 28424.97,E2 28424.97} C_VEL
LIN {X 0,Y 751.882,Z 320.565,A -85,B 0,C 180,E1 28422.669,E2 28422.669} C_VEL
LIN {X 0,Y 751.963,Z 320.565,A -85,B 0,C 180,E1 28419.845,E2 28419.845} C_VEL
LIN {X 0,Y 751.872,Z 320.567,A -85,B 0,C 180,E1 28417.15,E2 28417.15} C_VEL
LIN {X 0,Y 751.863,Z 320.563,A -85,B 0,C 180,E1 28414.898,E2 28414.898} C_VEL
LIN {X 0,Y 751.868,Z 320.566,A -85,B 0,C 180,E1 28412.604,E2 28412.604} C_VEL
LIN {X 0,Y 751.892,Z 320.566,A -85,B 0,C 180,E1 28410.262,E2 28410.262} C_VEL
LIN {X 0,Y 751.914,Z 320.565,A -85,B 0,C 180,E1 28407.233,E2 28407.233} C_VEL
LIN {X 0,Y 751.879,Z 320.565,A -85,B 0,C 180,E1 28404.738,E2 28404.738} C_VEL
LIN {X 0,Y 751.879,Z 320.565,A -85,B 0,C 180,E1 28402.477,E2 28402.477} C_VEL
LIN {X 0,Y 751.899,Z 320.567,A -85,B 0,C 180,E1 28400.112,E2 28400.112} C_VEL
LIN {X 0,Y 751.956,Z 320.563,A -85,B 0,C 180,E1 28397.196,E2 28397.196} C_VEL
LIN {X 0,Y 751.893,Z 320.566,A -85,B 0,C 180,E1 28394.537,E2 28394.537} C_VEL
LIN {X 0,Y 752.011,Z 320.791,A -85,B 0,C 180,E1 28393.425,E2 28393.425} C_VEL
LIN {X 0,Y 753.303,Z 324.603,A -85,B 0,C 180,E1 28393.077,E2 28393.077} C_VEL
LIN {X 0,Y 753.383,Z 351.247,A -85,B 0,C 180,E1 28391.342,E2 28391.342} C_VEL
LIN {X 0,Y 753.827,Z 354.251,A -85,B 0,C 180,E1 28391.275,E2 28391.275} C_VEL
LIN {X 0,Y 753.627,Z 564.448,A -85,B 0,C 180,E1 28388.726,E2 28388.726} C_VEL
LIN {X 0,Y 753.413,Z 790.832,A -85,B 0,C 180,E1 28386.078,E2 28386.078} C_VEL
LIN {X 0,Y 753.35,Z 832.024,A -85,B 0,C 180,E1 28385.573,E2 28385.573} C_VEL
LIN {X 0,Y 753.272,Z 858.362,A -85,B 0,C 180,E1 28385.103,E2 28385.103} C_VEL
LIN {X 0,Y 753.188,Z 884.936,A -85,B 0,C 180,E1 28384.475,E2 28384.475} C_VEL
LIN {X 0,Y 753.09,Z 910.679,A -85,B 0,C 180,E1 28383.709,E2 28383.709} C_VEL
LIN {X 0,Y 752.955,Z 937.222,A -85,B 0,C 180,E1 28382.761,E2 28382.761} C_VEL
LIN {X 0,Y 752.856,Z 958.681,A -85,B 0,C 180,E1 28381.866,E2 28381.866} C_VEL
LIN {X 0,Y 752.759,Z 977.618,A -85,B 0,C 180,E1 28380.978,E2 28380.978} C_VEL
LIN {X 0,Y 752.666,Z 996.701,A -85,B 0,C 180,E1 28379.984,E2 28379.984} C_VEL
LIN {X 0,Y 752.56,Z 1016.605,A -85,B 0,C 180,E1 28378.836,E2 28378.836} C_VEL
LIN {X 0,Y 752.414,Z 1040.409,A -85,B 0,C 180,E1 28377.288,E2 28377.288} C_VEL
LIN {X 0,Y 752.344,Z 1058.495,A -85,B 0,C 180,E1 28375.971,E2 28375.971} C_VEL
LIN {X 0,Y 752.262,Z 1076.352,A -85,B 0,C 180,E1 28374.542,E2 28374.542} C_VEL
LIN {X 0,Y 752.169,Z 1096.261,A -85,B 0,C 180,E1 28372.758,E2 28372.758} C_VEL
LIN {X 0,Y 752.095,Z 1111.284,A -85,B 0,C 180,E1 28371.257,E2 28371.257} C_VEL
LIN {X 0,Y 752.063,Z 1125.174,A -85,B 0,C 180,E1 28369.727,E2 28369.727} C_VEL
LIN {X 0,Y 752.008,Z 1141.334,A -85,B 0,C 180,E1 28367.727,E2 28367.727} C_VEL
LIN {X 0,Y 751.956,Z 1153.164,A -85,B 0,C 180,E1 28366.056,E2 28366.056} C_VEL
LIN {X 0,Y 751.954,Z 1163.123,A -85,B 0,C 180,E1 28364.477,E2 28364.477} C_VEL
LIN {X 0,Y 751.94,Z 1171.878,A -85,B 0,C 180,E1 28362.909,E2 28362.909} C_VEL
LIN {X 0,Y 751.931,Z 1179.498,A -85,B 0,C 180,E1 28361.35,E2 28361.35} C_VEL
LIN {X 0,Y 751.916,Z 1187.308,A -85,B 0,C 180,E1 28359.491,E2 28359.491} C_VEL
LIN {X 0,Y 751.911,Z 1194.032,A -85,B 0,C 180,E1 28357.488,E2 28357.488} C_VEL
LIN {X 0,Y 751.911,Z 1199.279,A -85,B 0,C 180,E1 28355.418,E2 28355.418} C_VEL
LIN {X 0,Y 751.914,Z 1202.788,A -85,B 0,C 180,E1 28353.355,E2 28353.355} C_VEL
LIN {X 0,Y 751.915,Z 1204.603,A -85,B 0,C 180,E1 28351.372,E2 28351.372} C_VEL
LIN {X 0,Y 751.889,Z 1204.849,A -85,B 0,C 180,E1 28349.467,E2 28349.467} C_VEL
LIN {X 0,Y 751.907,Z 1203.907,A -85,B 0,C 180,E1 28347.638,E2 28347.638} C_VEL
LIN {X 0,Y 751.907,Z 1201.054,A -85,B 0,C 180,E1 28345.5,E2 28345.5} C_VEL
LIN {X 0,Y 751.912,Z 1196.567,A -85,B 0,C 180,E1 28343.434,E2 28343.434} C_VEL
LIN {X 0,Y 751.92,Z 1190.63,A -85,B 0,C 180,E1 28341.435,E2 28341.435} C_VEL
LIN {X 0,Y 751.905,Z 1182.636,A -85,B 0,C 180,E1 28339.338,E2 28339.338} C_VEL
LIN {X 0,Y 751.935,Z 1173.113,A -85,B 0,C 180,E1 28337.326,E2 28337.326} C_VEL
LIN {X 0,Y 751.955,Z 1164.058,A -85,B 0,C 180,E1 28335.681,E2 28335.681} C_VEL
LIN {X 0,Y 751.954,Z 1154.214,A -85,B 0,C 180,E1 28334.103,E2 28334.103} C_VEL
LIN {X 0,Y 752.006,Z 1143.086,A -85,B 0,C 180,E1 28332.513,E2 28332.513} C_VEL
LIN {X 0,Y 752.066,Z 1127.932,A -85,B 0,C 180,E1 28330.587,E2 28330.587} C_VEL
LIN {X 0,Y 752.089,Z 1112.615,A -85,B 0,C 180,E1 28328.883,E2 28328.883} C_VEL
LIN {X 0,Y 752.166,Z 1097.974,A -85,B 0,C 180,E1 28327.408,E2 28327.408} C_VEL
LIN {X 0,Y 752.232,Z 1079.858,A -85,B 0,C 180,E1 28325.75,E2 28325.75} C_VEL
LIN {X 0,Y 752.346,Z 1060.164,A -85,B 0,C 180,E1 28324.157,E2 28324.157} C_VEL
LIN {X 0,Y 752.409,Z 1042.838,A -85,B 0,C 180,E1 28322.883,E2 28322.883} C_VEL
LIN {X 0,Y 752.521,Z 1022.266,A -85,B 0,C 180,E1 28321.511,E2 28321.511} C_VEL
LIN {X 0,Y 752.657,Z 998.635,A -85,B 0,C 180,E1 28320.121,E2 28320.121} C_VEL
LIN {X 0,Y 752.754,Z 979.253,A -85,B 0,C 180,E1 28319.103,E2 28319.103} C_VEL
LIN {X 0,Y 752.85,Z 960.434,A -85,B 0,C 180,E1 28318.213,E2 28318.213} C_VEL
LIN {X 0,Y 752.948,Z 940.596,A -85,B 0,C 180,E1 28317.375,E2 28317.375} C_VEL
LIN {X 0,Y 753.037,Z 920.034,A -85,B 0,C 180,E1 28316.608,E2 28316.608} C_VEL
LIN {X 0,Y 753.159,Z 894.911,A -85,B 0,C 180,E1 28315.802,E2 28315.802} C_VEL
LIN {X 0,Y 753.243,Z 867.434,A -85,B 0,C 180,E1 28315.094,E2 28315.094} C_VEL
LIN {X 0,Y 753.33,Z 841.908,A -85,B 0,C 180,E1 28314.586,E2 28314.586} C_VEL
LIN {X 0,Y 753.38,Z 814.909,A -85,B 0,C 180,E1 28314.198,E2 28314.198} C_VEL
LIN {X 0,Y 753.595,Z 589.646,A -85,B 0,C 180,E1 28311.573,E2 28311.573} C_VEL
LIN {X 0,Y 753.781,Z 383.723,A -85,B 0,C 180,E1 28309.087,E2 28309.087} C_VEL
LIN {X 0,Y 753.64,Z 352.252,A -85,B 0,C 180,E1 28308.688,E2 28308.688} C_VEL
LIN {X 0,Y 753.255,Z 350.368,A -85,B 0,C 180,E1 28308.621,E2 28308.621} C_VEL
LIN {X 0,Y 753.181,Z 323.915,A -85,B 0,C 180,E1 28306.869,E2 28306.869} C_VEL
LIN {X 0,Y 751.979,Z 320.566,A -85,B 0,C 180,E1 28306.553,E2 28306.553} C_VEL
LIN {X 0,Y 751.897,Z 320.566,A -85,B 0,C 180,E1 28303.855,E2 28303.855} C_VEL
LIN {X 0,Y 751.887,Z 320.565,A -85,B 0,C 180,E1 28301.473,E2 28301.473} C_VEL
LIN {X 0,Y 751.914,Z 320.563,A -85,B 0,C 180,E1 28298.976,E2 28298.976} C_VEL
LIN {X 0,Y 751.911,Z 320.565,A -85,B 0,C 180,E1 28295.905,E2 28295.905} C_VEL
LIN {X 0,Y 751.881,Z 320.565,A -85,B 0,C 180,E1 28293.497,E2 28293.497} C_VEL
LIN {X 0,Y 751.877,Z 320.564,A -85,B 0,C 180,E1 28291.232,E2 28291.232} C_VEL
LIN {X 0,Y 751.883,Z 320.565,A -85,B 0,C 180,E1 28288.951,E2 28288.951} C_VEL
LIN {X 0,Y 751.973,Z 320.564,A -85,B 0,C 180,E1 28286.197,E2 28286.197} C_VEL
LIN {X 0,Y 751.88,Z 320.566,A -85,B 0,C 180,E1 28283.426,E2 28283.426} C_VEL
LIN {X 0,Y 751.868,Z 320.564,A -85,B 0,C 180,E1 28281.206,E2 28281.206} C_VEL
LIN {X 0,Y 751.864,Z 320.566,A -85,B 0,C 180,E1 28278.999,E2 28278.999} C_VEL
LIN {X 0,Y 751.866,Z 320.564,A -85,B 0,C 180,E1 28276.766,E2 28276.766} C_VEL
LIN {X 0,Y 751.913,Z 320.566,A -85,B 0,C 180,E1 28274.242,E2 28274.242} C_VEL
LIN {X 0,Y 751.887,Z 320.564,A -85,B 0,C 180,E1 28271.273,E2 28271.273} C_VEL
LIN {X 0,Y 751.868,Z 320.566,A -85,B 0,C 180,E1 28268.951,E2 28268.951} C_VEL
LIN {X 0,Y 751.869,Z 320.564,A -85,B 0,C 180,E1 28266.721,E2 28266.721} C_VEL
LIN {X 0,Y 751.878,Z 320.565,A -85,B 0,C 180,E1 28264.424,E2 28264.424} C_VEL
LIN {X 0,Y 751.973,Z 320.565,A -85,B 0,C 180,E1 28261.676,E2 28261.676} C_VEL
LIN {X 0,Y 751.889,Z 320.564,A -85,B 0,C 180,E1 28258.857,E2 28258.857} C_VEL
LIN {X 0,Y 751.878,Z 320.564,A -85,B 0,C 180,E1 28256.493,E2 28256.493} C_VEL
LIN {X 0,Y 751.88,Z 320.562,A -85,B 0,C 180,E1 28254.484,E2 28254.484} C_VEL
LIN {X 0,Y 750.886,Z 320.691,A -85,B 0,C 180,E1 28253.897,E2 28253.897} C_VEL
LIN {X 0,Y 744.474,Z 321.49,A -85,B 0,C 180,E1 28252.253,E2 28252.253} C_VEL
LIN {X 0,Y 743.981,Z 321.555,A -85,B 0,C 180,E1 28251.826,E2 28251.826} C_VEL
LIN {X 0,Y 743.972,Z 321.549,A -85,B 0,C 180,E1 28248.762,E2 28248.762} C_VEL
LIN {X 0,Y 743.951,Z 321.552,A -85,B 0,C 180,E1 28246.317,E2 28246.317} C_VEL
LIN {X 0,Y 743.96,Z 321.548,A -85,B 0,C 180,E1 28243.927,E2 28243.927} C_VEL
LIN {X 0,Y 744.041,Z 321.549,A -85,B 0,C 180,E1 28241.095,E2 28241.095} C_VEL
LIN {X 0,Y 743.964,Z 321.551,A -85,B 0,C 180,E1 28238.309,E2 28238.309} C_VEL
LIN {X 0,Y 743.961,Z 321.551,A -85,B 0,C 180,E1 28235.862,E2 28235.862} C_VEL
LIN {X 0,Y 744.034,Z 321.555,A -85,B 0,C 180,E1 28233.157,E2 28233.157} C_VEL
LIN {X 0,Y 743.98,Z 321.549,A -85,B 0,C 180,E1 28230.249,E2 28230.249} C_VEL
LIN {X 0,Y 743.968,Z 321.552,A -85,B 0,C 180,E1 28227.71,E2 28227.71} C_VEL
LIN {X 0,Y 744.03,Z 321.556,A -85,B 0,C 180,E1 28224.981,E2 28224.981} C_VEL
LIN {X 0,Y 743.984,Z 321.551,A -85,B 0,C 180,E1 28222.009,E2 28222.009} C_VEL
LIN {X 0,Y 743.98,Z 321.557,A -85,B 0,C 180,E1 28219.405,E2 28219.405} C_VEL
LIN {X 0,Y 744.012,Z 321.722,A -85,B 0,C 180,E1 28219.254,E2 28219.254} C_VEL
LIN {X 0,Y 745.451,Z 325.207,A -85,B 0,C 180,E1 28218.909,E2 28218.909} C_VEL
LIN {X 0,Y 746.66,Z 328.716,A -85,B 0,C 180,E1 28218.582,E2 28218.582} C_VEL
LIN {X 0,Y 746.693,Z 341.413,A -85,B 0,C 180,E1 28217.748,E2 28217.748} C_VEL
LIN {X 0,Y 747.814,Z 346.17,A -85,B 0,C 180,E1 28217.611,E2 28217.611} C_VEL
LIN {X 0,Y 747.369,Z 559.772,A -85,B 0,C 180,E1 28215.002,E2 28215.002} C_VEL
LIN {X 0,Y 746.925,Z 786.654,A -85,B 0,C 180,E1 28212.328,E2 28212.328} C_VEL
LIN {X 0,Y 746.818,Z 823.691,A -85,B 0,C 180,E1 28211.863,E2 28211.863} C_VEL
LIN {X 0,Y 746.653,Z 850.377,A -85,B 0,C 180,E1 28211.373,E2 28211.373} C_VEL
LIN {X 0,Y 746.483,Z 876.497,A -85,B 0,C 180,E1 28210.741,E2 28210.741} C_VEL
LIN {X 0,Y 746.276,Z 904.269,A -85,B 0,C 180,E1 28209.899,E2 28209.899} C_VEL
LIN {X 0,Y 746.007,Z 929.232,A -85,B 0,C 180,E1 28208.978,E2 28208.978} C_VEL
LIN {X 0,Y 745.817,Z 949.417,A -85,B 0,C 180,E1 28208.124,E2 28208.124} C_VEL
LIN {X 0,Y 745.615,Z 968.956,A -85,B 0,C 180,E1 28207.196,E2 28207.196} C_VEL
LIN {X 0,Y 745.425,Z 989.105,A -85,B 0,C 180,E1 28206.127,E2 28206.127} C_VEL
LIN {X 0,Y 745.14,Z 1013.418,A -85,B 0,C 180,E1 28204.677,E2 28204.677} C_VEL
LIN {X 0,Y 744.944,Z 1033.178,A -85,B 0,C 180,E1 28203.342,E2 28203.342} C_VEL
LIN {X 0,Y 744.775,Z 1050.883,A -85,B 0,C 180,E1 28202.025,E2 28202.025} C_VEL
LIN {X 0,Y 744.561,Z 1071.457,A -85,B 0,C 180,E1 28200.326,E2 28200.326} C_VEL
LIN {X 0,Y 744.427,Z 1088.54,A -85,B 0,C 180,E1 28198.74,E2 28198.74} C_VEL
LIN {X 0,Y 744.307,Z 1103.818,A -85,B 0,C 180,E1 28197.177,E2 28197.177} C_VEL
LIN {X 0,Y 744.173,Z 1120.947,A -85,B 0,C 180,E1 28195.209,E2 28195.209} C_VEL
LIN {X 0,Y 744.085,Z 1133.9,A -85,B 0,C 180,E1 28193.521,E2 28193.521} C_VEL
LIN {X 0,Y 744.026,Z 1144.494,A -85,B 0,C 180,E1 28191.984,E2 28191.984} C_VEL
LIN {X 0,Y 744,Z 1154.418,A -85,B 0,C 180,E1 28190.369,E2 28190.369} C_VEL
LIN {X 0,Y 743.966,Z 1164.544,A -85,B 0,C 180,E1 28188.492,E2 28188.492} C_VEL
LIN {X 0,Y 743.936,Z 1174.67,A -85,B 0,C 180,E1 28186.234,E2 28186.234} C_VEL
LIN {X 0,Y 743.921,Z 1181.845,A -85,B 0,C 180,E1 28184.238,E2 28184.238} C_VEL
LIN {X 0,Y 743.914,Z 1187.602,A -85,B 0,C 180,E1 28182.182,E2 28182.182} C_VEL
LIN {X 0,Y 743.91,Z 1191.766,A -85,B 0,C 180,E1 28180.063,E2 28180.063} C_VEL
LIN {X 0,Y 743.914,Z 1194.156,A -85,B 0,C 180,E1 28178.035,E2 28178.035} C_VEL
LIN {X 0,Y 743.897,Z 1194.957,A -85,B 0,C 180,E1 28175.785,E2 28175.785} C_VEL
LIN {X 0,Y 743.911,Z 1194.027,A -85,B 0,C 180,E1 28173.699,E2 28173.699} C_VEL
LIN {X 0,Y 743.914,Z 1191.394,A -85,B 0,C 180,E1 28171.617,E2 28171.617} C_VEL
LIN {X 0,Y 743.917,Z 1187.316,A -85,B 0,C 180,E1 28169.615,E2 28169.615} C_VEL
LIN {X 0,Y 743.925,Z 1181.169,A -85,B 0,C 180,E1 28167.458,E2 28167.458} C_VEL
LIN {X 0,Y 743.915,Z 1173.44,A -85,B 0,C 180,E1 28165.374,E2 28165.374} C_VEL
LIN {X 0,Y 743.972,Z 1163.448,A -85,B 0,C 180,E1 28163.207,E2 28163.207} C_VEL
LIN {X 0,Y 743.988,Z 1154.17,A -85,B 0,C 180,E1 28161.498,E2 28161.498} C_VEL
LIN {X 0,Y 744.033,Z 1144.571,A -85,B 0,C 180,E1 28159.938,E2 28159.938} C_VEL
LIN {X 0,Y 744.086,Z 1133.775,A -85,B 0,C 180,E1 28158.371,E2 28158.371} C_VEL
LIN {X 0,Y 744.185,Z 1120.143,A -85,B 0,C 180,E1 28156.6,E2 28156.6} C_VEL
LIN {X 0,Y 744.296,Z 1103.532,A -85,B 0,C 180,E1 28154.703,E2 28154.703} C_VEL
LIN {X 0,Y 744.428,Z 1089.003,A -85,B 0,C 180,E1 28153.215,E2 28153.215} C_VEL
LIN {X 0,Y 744.535,Z 1072.577,A -85,B 0,C 180,E1 28151.684,E2 28151.684} C_VEL
LIN {X 0,Y 744.766,Z 1051.81,A -85,B 0,C 180,E1 28149.957,E2 28149.957} C_VEL
LIN {X 0,Y 744.921,Z 1034.143,A -85,B 0,C 180,E1 28148.636,E2 28148.636} C_VEL
LIN {X 0,Y 745.117,Z 1015.168,A -85,B 0,C 180,E1 28147.348,E2 28147.348} C_VEL
LIN {X 0,Y 745.418,Z 990.34,A -85,B 0,C 180,E1 28145.85,E2 28145.85} C_VEL
LIN {X 0,Y 745.616,Z 969.82,A -85,B 0,C 180,E1 28144.758,E2 28144.758} C_VEL
LIN {X 0,Y 745.81,Z 950.316,A -85,B 0,C 180,E1 28143.827,E2 28143.827} C_VEL
LIN {X 0,Y 746.003,Z 930.294,A -85,B 0,C 180,E1 28142.976,E2 28142.976} C_VEL
LIN {X 0,Y 746.196,Z 907.325,A -85,B 0,C 180,E1 28142.118,E2 28142.118} C_VEL
LIN {X 0,Y 746.456,Z 878.108,A -85,B 0,C 180,E1 28141.213,E2 28141.213} C_VEL
LIN {X 0,Y 746.659,Z 852.315,A -85,B 0,C 180,E1 28140.58,E2 28140.58} C_VEL
LIN {X 0,Y 746.81,Z 825.054,A -85,B 0,C 180,E1 28140.067,E2 28140.067} C_VEL
LIN {X 0,Y 746.911,Z 791.046,A -85,B 0,C 180,E1 28139.633,E2 28139.633} C_VEL
LIN {X 0,Y 747.354,Z 563.403,A -85,B 0,C 180,E1 28136.951,E2 28136.951} C_VEL
LIN {X 0,Y 747.815,Z 349.264,A -85,B 0,C 180,E1 28134.338,E2 28134.338} C_VEL
LIN {X 0,Y 747.618,Z 344.609,A -85,B 0,C 180,E1 28134.266,E2 28134.266} C_VEL
LIN {X 0,Y 746.573,Z 340.503,A -85,B 0,C 180,E1 28134.124,E2 28134.124} C_VEL
LIN {X 0,Y 746.603,Z 328.143,A -85,B 0,C 180,E1 28133.285,E2 28133.285} C_VEL
LIN {X 0,Y 744.01,Z 321.555,A -85,B 0,C 180,E1 28132.643,E2 28132.643} C_VEL
LIN {X 0,Y 744.032,Z 321.546,A -85,B 0,C 180,E1 28129.759,E2 28129.759} C_VEL
LIN {X 0,Y 744.026,Z 321.556,A -85,B 0,C 180,E1 28126.84,E2 28126.84} C_VEL
LIN {X 0,Y 744.02,Z 321.545,A -85,B 0,C 180,E1 28123.904,E2 28123.904} C_VEL
LIN {X 0,Y 744.033,Z 321.556,A -85,B 0,C 180,E1 28120.835,E2 28120.835} C_VEL
LIN {X 0,Y 743.999,Z 321.547,A -85,B 0,C 180,E1 28117.99,E2 28117.99} C_VEL
LIN {X 0,Y 744.029,Z 321.548,A -85,B 0,C 180,E1 28115.207,E2 28115.207} C_VEL
LIN {X 0,Y 743.998,Z 321.552,A -85,B 0,C 180,E1 28112.337,E2 28112.337} C_VEL
LIN {X 0,Y 744.009,Z 321.546,A -85,B 0,C 180,E1 28109.553,E2 28109.553} C_VEL
LIN {X 0,Y 744.018,Z 321.551,A -85,B 0,C 180,E1 28106.488,E2 28106.488} C_VEL
LIN {X 0,Y 743.982,Z 321.549,A -85,B 0,C 180,E1 28103.761,E2 28103.761} C_VEL
LIN {X 0,Y 744.036,Z 321.545,A -85,B 0,C 180,E1 28100.936,E2 28100.936} C_VEL
LIN {X 0,Y 743.988,Z 321.553,A -85,B 0,C 180,E1 28098.087,E2 28098.087} C_VEL
LIN {X 0,Y 743.976,Z 321.548,A -85,B 0,C 180,E1 28095.502,E2 28095.502} C_VEL
LIN {X 0,Y 744.037,Z 321.544,A -85,B 0,C 180,E1 28092.653,E2 28092.653} C_VEL
LIN {X 0,Y 743.973,Z 321.552,A -85,B 0,C 180,E1 28089.828,E2 28089.828} C_VEL
LIN {X 0,Y 743.967,Z 321.55,A -85,B 0,C 180,E1 28087.316,E2 28087.316} C_VEL
LIN {X 0,Y 744.04,Z 321.548,A -85,B 0,C 180,E1 28084.548,E2 28084.548} C_VEL
LIN {X 0,Y 743.966,Z 321.552,A -85,B 0,C 180,E1 28081.694,E2 28081.694} C_VEL
LIN {X 0,Y 743.952,Z 321.552,A -85,B 0,C 180,E1 28079.307,E2 28079.307} C_VEL
LIN {X 0,Y 743.974,Z 321.551,A -85,B 0,C 180,E1 28076.841,E2 28076.841} C_VEL
LIN {X 0,Y 743.988,Z 321.555,A -85,B 0,C 180,E1 28073.828,E2 28073.828} C_VEL
LIN {X 0,Y 743.945,Z 321.553,A -85,B 0,C 180,E1 28071.342,E2 28071.342} C_VEL
LIN {X 0,Y 743.939,Z 321.554,A -85,B 0,C 180,E1 28069.076,E2 28069.076} C_VEL
LIN {X 0,Y 743.951,Z 321.549,A -85,B 0,C 180,E1 28066.713,E2 28066.713} C_VEL
LIN {X 0,Y 744.016,Z 321.556,A -85,B 0,C 180,E1 28063.848,E2 28063.848} C_VEL
LIN {X 0,Y 743.935,Z 321.552,A -85,B 0,C 180,E1 28061.181,E2 28061.181} C_VEL
LIN {X 0,Y 743.926,Z 321.554,A -85,B 0,C 180,E1 28058.969,E2 28058.969} C_VEL
LIN {X 0,Y 743.923,Z 321.556,A -85,B 0,C 180,E1 28056.808,E2 28056.808} C_VEL
LIN {X 0,Y 743.933,Z 321.55,A -85,B 0,C 180,E1 28054.526,E2 28054.526} C_VEL
LIN {X 0,Y 744.035,Z 321.555,A -85,B 0,C 180,E1 28051.768,E2 28051.768} C_VEL
LIN {X 0,Y 743.945,Z 321.553,A -85,B 0,C 180,E1 28049.018,E2 28049.018} C_VEL
LIN {X 0,Y 743.937,Z 321.555,A -85,B 0,C 180,E1 28046.719,E2 28046.719} C_VEL
LIN {X 0,Y 743.942,Z 321.555,A -85,B 0,C 180,E1 28044.404,E2 28044.404} C_VEL
LIN {X 0,Y 744.018,Z 321.557,A -85,B 0,C 180,E1 28041.705,E2 28041.705} C_VEL
LIN {X 0,Y 743.96,Z 321.553,A -85,B 0,C 180,E1 28038.809,E2 28038.809} C_VEL
LIN {X 0,Y 743.949,Z 321.556,A -85,B 0,C 180,E1 28036.41,E2 28036.41} C_VEL
LIN {X 0,Y 743.98,Z 321.631,A -85,B 0,C 180,E1 28033.956,E2 28033.956} C_VEL
LIN {X 0,Y 745.067,Z 324.654,A -85,B 0,C 180,E1 28033.668,E2 28033.668} C_VEL
LIN {X 0,Y 746.726,Z 328.287,A -85,B 0,C 180,E1 28033.3,E2 28033.3} C_VEL
LIN {X 0,Y 746.773,Z 351.26,A -85,B 0,C 180,E1 28031.789,E2 28031.789} C_VEL
LIN {X 0,Y 747.795,Z 355.973,A -85,B 0,C 180,E1 28031.66,E2 28031.66} C_VEL
LIN {X 0,Y 747.37,Z 566.135,A -85,B 0,C 180,E1 28029.091,E2 28029.091} C_VEL
LIN {X 0,Y 746.935,Z 792.082,A -85,B 0,C 180,E1 28026.426,E2 28026.426} C_VEL
LIN {X 0,Y 746.817,Z 832.608,A -85,B 0,C 180,E1 28025.924,E2 28025.924} C_VEL
LIN {X 0,Y 746.661,Z 859.16,A -85,B 0,C 180,E1 28025.443,E2 28025.443} C_VEL
LIN {X 0,Y 746.494,Z 885.287,A -85,B 0,C 180,E1 28024.818,E2 28024.818} C_VEL
LIN {X 0,Y 746.294,Z 912.15,A -85,B 0,C 180,E1 28024.012,E2 28024.012} C_VEL
LIN {X 0,Y 746.013,Z 938.345,A -85,B 0,C 180,E1 28023.059,E2 28023.059} C_VEL
LIN {X 0,Y 745.813,Z 959.678,A -85,B 0,C 180,E1 28022.157,E2 28022.157} C_VEL
LIN {X 0,Y 745.617,Z 979.491,A -85,B 0,C 180,E1 28021.214,E2 28021.214} C_VEL
LIN {X 0,Y 745.41,Z 1001.034,A -85,B 0,C 180,E1 28020.067,E2 28020.067} C_VEL
LIN {X 0,Y 745.121,Z 1024.908,A -85,B 0,C 180,E1 28018.624,E2 28018.624} C_VEL
LIN {X 0,Y 744.926,Z 1043.434,A -85,B 0,C 180,E1 28017.369,E2 28017.369} C_VEL
LIN {X 0,Y 744.78,Z 1061.263,A -85,B 0,C 180,E1 28016.04,E2 28016.04} C_VEL
LIN {X 0,Y 744.534,Z 1082.647,A -85,B 0,C 180,E1 28014.264,E2 28014.264} C_VEL
LIN {X 0,Y 744.424,Z 1098.823,A -85,B 0,C 180,E1 28012.758,E2 28012.758} C_VEL
LIN {X 0,Y 744.287,Z 1114.951,A -85,B 0,C 180,E1 28011.102,E2 28011.102} C_VEL
LIN {X 0,Y 744.155,Z 1131.862,A -85,B 0,C 180,E1 28009.138,E2 28009.138} C_VEL
LIN {X 0,Y 744.097,Z 1144.247,A -85,B 0,C 180,E1 28007.518,E2 28007.518} C_VEL
LIN {X 0,Y 744.02,Z 1154.733,A -85,B 0,C 180,E1 28005.992,E2 28005.992} C_VEL
LIN {X 0,Y 743.999,Z 1164.521,A -85,B 0,C 180,E1 28004.396,E2 28004.396} C_VEL
LIN {X 0,Y 743.962,Z 1174.753,A -85,B 0,C 180,E1 28002.497,E2 28002.497} C_VEL
LIN {X 0,Y 743.933,Z 1184.911,A -85,B 0,C 180,E1 28000.219,E2 28000.219} C_VEL
LIN {X 0,Y 743.922,Z 1191.891,A -85,B 0,C 180,E1 27998.269,E2 27998.269} C_VEL
LIN {X 0,Y 743.916,Z 1197.734,A -85,B 0,C 180,E1 27996.173,E2 27996.173} C_VEL
LIN {X 0,Y 743.91,Z 1201.927,A -85,B 0,C 180,E1 27994.008,E2 27994.008} C_VEL
LIN {X 0,Y 743.912,Z 1204.212,A -85,B 0,C 180,E1 27992.003,E2 27992.003} C_VEL
LIN {X 0,Y 743.898,Z 1204.939,A -85,B 0,C 180,E1 27989.769,E2 27989.769} C_VEL
LIN {X 0,Y 743.908,Z 1203.979,A -85,B 0,C 180,E1 27987.689,E2 27987.689} C_VEL
LIN {X 0,Y 743.912,Z 1201.304,A -85,B 0,C 180,E1 27985.606,E2 27985.606} C_VEL
LIN {X 0,Y 743.919,Z 1197.153,A -85,B 0,C 180,E1 27983.595,E2 27983.595} C_VEL
LIN {X 0,Y 743.924,Z 1191.155,A -85,B 0,C 180,E1 27981.498,E2 27981.498} C_VEL
LIN {X 0,Y 743.919,Z 1183.319,A -85,B 0,C 180,E1 27979.39,E2 27979.39} C_VEL
LIN {X 0,Y 743.966,Z 1173.524,A -85,B 0,C 180,E1 27977.267,E2 27977.267} C_VEL
LIN {X 0,Y 743.999,Z 1164.525,A -85,B 0,C 180,E1 27975.604,E2 27975.604} C_VEL
LIN {X 0,Y 744.02,Z 1154.738,A -85,B 0,C 180,E1 27974.009,E2 27974.009} C_VEL
LIN {X 0,Y 744.097,Z 1144.252,A -85,B 0,C 180,E1 27972.483,E2 27972.483} C_VEL
LIN {X 0,Y 744.155,Z 1131.867,A -85,B 0,C 180,E1 27970.862,E2 27970.862} C_VEL
LIN {X 0,Y 744.287,Z 1114.957,A -85,B 0,C 180,E1 27968.898,E2 27968.898} C_VEL
LIN {X 0,Y 744.424,Z 1098.83,A -85,B 0,C 180,E1 27967.243,E2 27967.243} C_VEL
LIN {X 0,Y 744.541,Z 1082.149,A -85,B 0,C 180,E1 27965.691,E2 27965.691} C_VEL
LIN {X 0,Y 744.78,Z 1061.272,A -85,B 0,C 180,E1 27963.96,E2 27963.96} C_VEL
LIN {X 0,Y 744.926,Z 1043.443,A -85,B 0,C 180,E1 27962.631,E2 27962.631} C_VEL
LIN {X 0,Y 745.123,Z 1024.605,A -85,B 0,C 180,E1 27961.356,E2 27961.356} C_VEL
LIN {X 0,Y 745.415,Z 1000.243,A -85,B 0,C 180,E1 27959.89,E2 27959.89} C_VEL
LIN {X 0,Y 745.617,Z 979.504,A -85,B 0,C 180,E1 27958.787,E2 27958.787} C_VEL
LIN {X 0,Y 745.814,Z 959.695,A -85,B 0,C 180,E1 27957.844,E2 27957.844} C_VEL
LIN {X 0,Y 746.015,Z 938.363,A -85,B 0,C 180,E1 27956.942,E2 27956.942} C_VEL
LIN {X 0,Y 746.298,Z 911.438,A -85,B 0,C 180,E1 27955.966,E2 27955.966} C_VEL
LIN {X 0,Y 746.495,Z 885.162,A -85,B 0,C 180,E1 27955.178,E2 27955.178} C_VEL
LIN {X 0,Y 746.663,Z 858.718,A -85,B 0,C 180,E1 27954.547,E2 27954.547} C_VEL
LIN {X 0,Y 746.819,Z 832.262,A -85,B 0,C 180,E1 27954.071,E2 27954.071} C_VEL
LIN {X 0,Y 746.94,Z 790.253,A -85,B 0,C 180,E1 27953.553,E2 27953.553} C_VEL
LIN {X 0,Y 747.379,Z 563.128,A -85,B 0,C 180,E1 27950.873,E2 27950.873} C_VEL
LIN {X 0,Y 747.798,Z 355.17,A -85,B 0,C 180,E1 27948.33,E2 27948.33} C_VEL
LIN {X 0,Y 746.643,Z 350.368,A -85,B 0,C 180,E1 27948.172,E2 27948.172} C_VEL
LIN {X 0,Y 746.726,Z 328.287,A -85,B 0,C 180,E1 27946.7,E2 27946.7} C_VEL
LIN {X 0,Y 745.067,Z 324.653,A -85,B 0,C 180,E1 27946.332,E2 27946.332} C_VEL
LIN {X 0,Y 743.97,Z 321.56,A -85,B 0,C 180,E1 27946.025,E2 27946.025} C_VEL
LIN {X 0,Y 743.95,Z 321.556,A -85,B 0,C 180,E1 27943.58,E2 27943.58} C_VEL
LIN {X 0,Y 743.971,Z 321.553,A -85,B 0,C 180,E1 27941.088,E2 27941.088} C_VEL
LIN {X 0,Y 743.986,Z 321.555,A -85,B 0,C 180,E1 27938.043,E2 27938.043} C_VEL
LIN {X 0,Y 743.943,Z 321.553,A -85,B 0,C 180,E1 27935.495,E2 27935.495} C_VEL
LIN {X 0,Y 743.945,Z 321.553,A -85,B 0,C 180,E1 27933.142,E2 27933.142} C_VEL
LIN {X 0,Y 744.006,Z 321.551,A -85,B 0,C 180,E1 27930.522,E2 27930.522} C_VEL
LIN {X 0,Y 743.955,Z 321.553,A -85,B 0,C 180,E1 27927.625,E2 27927.625} C_VEL
LIN {X 0,Y 743.933,Z 321.554,A -85,B 0,C 180,E1 27925.24,E2 27925.24} C_VEL
LIN {X 0,Y 743.932,Z 321.554,A -85,B 0,C 180,E1 27922.977,E2 27922.977} C_VEL
LIN {X 0,Y 743.949,Z 321.552,A -85,B 0,C 180,E1 27920.618,E2 27920.618} C_VEL
LIN {X 0,Y 743.97,Z 321.552,A -85,B 0,C 180,E1 27917.602,E2 27917.602} C_VEL
LIN {X 0,Y 743.927,Z 321.555,A -85,B 0,C 180,E1 27915.115,E2 27915.115} C_VEL
LIN {X 0,Y 743.924,Z 321.555,A -85,B 0,C 180,E1 27912.813,E2 27912.813} C_VEL
LIN {X 0,Y 743.936,Z 321.552,A -85,B 0,C 180,E1 27910.532,E2 27910.532} C_VEL
LIN {X 0,Y 744.034,Z 321.553,A -85,B 0,C 180,E1 27907.723,E2 27907.723} C_VEL
LIN {X 0,Y 743.94,Z 321.552,A -85,B 0,C 180,E1 27904.935,E2 27904.935} C_VEL
LIN {X 0,Y 743.934,Z 321.555,A -85,B 0,C 180,E1 27902.619,E2 27902.619} C_VEL
LIN {X 0,Y 743.945,Z 321.551,A -85,B 0,C 180,E1 27900.308,E2 27900.308} C_VEL
LIN {X 0,Y 744.036,Z 321.554,A -85,B 0,C 180,E1 27897.535,E2 27897.535} C_VEL
LIN {X 0,Y 743.952,Z 321.548,A -85,B 0,C 180,E1 27894.756,E2 27894.756} C_VEL
LIN {X 0,Y 743.944,Z 321.553,A -85,B 0,C 180,E1 27892.431,E2 27892.431} C_VEL
LIN {X 0,Y 743.981,Z 321.555,A -85,B 0,C 180,E1 27891.826,E2 27891.826} C_VEL
LIN {X 0,Y 743.057,Z 321.679,A -85,B 0,C 180,E1 27891.233,E2 27891.233} C_VEL
LIN {X 0,Y 736.566,Z 322.484,A -85,B 0,C 180,E1 27889.529,E2 27889.529} C_VEL
LIN {X 0,Y 736.087,Z 322.537,A -85,B 0,C 180,E1 27889.14,E2 27889.14} C_VEL
LIN {X 0,Y 736.015,Z 322.541,A -85,B 0,C 180,E1 27886.407,E2 27886.407} C_VEL
LIN {X 0,Y 736.018,Z 322.535,A -85,B 0,C 180,E1 27883.991,E2 27883.991} C_VEL
LIN {X 0,Y 736.099,Z 322.54,A -85,B 0,C 180,E1 27881.219,E2 27881.219} C_VEL
LIN {X 0,Y 736.031,Z 322.539,A -85,B 0,C 180,E1 27878.398,E2 27878.398} C_VEL
LIN {X 0,Y 736.021,Z 322.54,A -85,B 0,C 180,E1 27875.909,E2 27875.909} C_VEL
LIN {X 0,Y 736.091,Z 322.544,A -85,B 0,C 180,E1 27873.181,E2 27873.181} C_VEL
LIN {X 0,Y 736.041,Z 322.538,A -85,B 0,C 180,E1 27870.232,E2 27870.232} C_VEL
LIN {X 0,Y 736.03,Z 322.541,A -85,B 0,C 180,E1 27867.731,E2 27867.731} C_VEL
LIN {X 0,Y 736.09,Z 322.545,A -85,B 0,C 180,E1 27864.993,E2 27864.993} C_VEL
LIN {X 0,Y 736.047,Z 322.541,A -85,B 0,C 180,E1 27862.02,E2 27862.02} C_VEL
LIN {X 0,Y 736.068,Z 322.762,A -85,B 0,C 180,E1 27859.766,E2 27859.766} C_VEL
LIN {X 0,Y 737.561,Z 326.332,A -85,B 0,C 180,E1 27859.404,E2 27859.404} C_VEL
LIN {X 0,Y 740.063,Z 332.22,A -85,B 0,C 180,E1 27858.811,E2 27858.811} C_VEL
LIN {X 0,Y 740.069,Z 341.367,A -85,B 0,C 180,E1 27858.208,E2 27858.208} C_VEL
LIN {X 0,Y 741.818,Z 348.265,A -85,B 0,C 180,E1 27857.998,E2 27857.998} C_VEL
LIN {X 0,Y 741.136,Z 562.652,A -85,B 0,C 180,E1 27855.359,E2 27855.359} C_VEL
LIN {X 0,Y 740.464,Z 789.772,A -85,B 0,C 180,E1 27852.66,E2 27852.66} C_VEL
LIN {X 0,Y 740.309,Z 824.928,A -85,B 0,C 180,E1 27852.209,E2 27852.209} C_VEL
LIN {X 0,Y 740.062,Z 852.202,A -85,B 0,C 180,E1 27851.696,E2 27851.696} C_VEL
LIN {X 0,Y 739.79,Z 878.146,A -85,B 0,C 180,E1 27851.055,E2 27851.055} C_VEL
LIN {X 0,Y 739.427,Z 906.729,A -85,B 0,C 180,E1 27850.166,E2 27850.166} C_VEL
LIN {X 0,Y 739.082,Z 930.335,A -85,B 0,C 180,E1 27849.282,E2 27849.282} C_VEL
LIN {X 0,Y 738.791,Z 950.781,A -85,B 0,C 180,E1 27848.404,E2 27848.404} C_VEL
LIN {X 0,Y 738.488,Z 970.771,A -85,B 0,C 180,E1 27847.439,E2 27847.439} C_VEL
LIN {X 0,Y 738.154,Z 994.298,A -85,B 0,C 180,E1 27846.164,E2 27846.164} C_VEL
LIN {X 0,Y 737.731,Z 1016.595,A -85,B 0,C 180,E1 27844.78,E2 27844.78} C_VEL
LIN {X 0,Y 737.47,Z 1034.626,A -85,B 0,C 180,E1 27843.538,E2 27843.538} C_VEL
LIN {X 0,Y 737.203,Z 1054.548,A -85,B 0,C 180,E1 27842.026,E2 27842.026} C_VEL
LIN {X 0,Y 736.867,Z 1074.245,A -85,B 0,C 180,E1 27840.342,E2 27840.342} C_VEL
LIN {X 0,Y 736.688,Z 1090.003,A -85,B 0,C 180,E1 27838.849,E2 27838.849} C_VEL
LIN {X 0,Y 736.498,Z 1107.184,A -85,B 0,C 180,E1 27837.05,E2 27837.05} C_VEL
LIN {X 0,Y 736.296,Z 1123.058,A -85,B 0,C 180,E1 27835.153,E2 27835.153} C_VEL
LIN {X 0,Y 736.183,Z 1134.593,A -85,B 0,C 180,E1 27833.619,E2 27833.619} C_VEL
LIN {X 0,Y 736.092,Z 1145.418,A -85,B 0,C 180,E1 27832.018,E2 27832.018} C_VEL
LIN {X 0,Y 736.044,Z 1156.526,A -85,B 0,C 180,E1 27830.165,E2 27830.165} C_VEL
LIN {X 0,Y 735.95,Z 1167.3,A -85,B 0,C 180,E1 27828.045,E2 27828.045} C_VEL
LIN {X 0,Y 735.947,Z 1175.681,A -85,B 0,C 180,E1 27826.09,E2 27826.09} C_VEL
LIN {X 0,Y 735.925,Z 1182.881,A -85,B 0,C 180,E1 27823.995,E2 27823.995} C_VEL
LIN {X 0,Y 735.911,Z 1188.342,A -85,B 0,C 180,E1 27821.918,E2 27821.918} C_VEL
LIN {X 0,Y 735.906,Z 1192.157,A -85,B 0,C 180,E1 27819.857,E2 27819.857} C_VEL
LIN {X 0,Y 735.904,Z 1194.392,A -85,B 0,C 180,E1 27817.73,E2 27817.73} C_VEL
LIN {X 0,Y 735.891,Z 1194.885,A -85,B 0,C 180,E1 27815.536,E2 27815.536} C_VEL
LIN {X 0,Y 735.907,Z 1193.945,A -85,B 0,C 180,E1 27813.583,E2 27813.583} C_VEL
LIN {X 0,Y 735.907,Z 1191.124,A -85,B 0,C 180,E1 27811.401,E2 27811.401} C_VEL
LIN {X 0,Y 735.916,Z 1186.895,A -85,B 0,C 180,E1 27809.377,E2 27809.377} C_VEL
LIN {X 0,Y 735.932,Z 1180.874,A -85,B 0,C 180,E1 27807.274,E2 27807.274} C_VEL
LIN {X 0,Y 735.942,Z 1172.762,A -85,B 0,C 180,E1 27805.09,E2 27805.09} C_VEL
LIN {X 0,Y 735.991,Z 1163.389,A -85,B 0,C 180,E1 27803.055,E2 27803.055} C_VEL
LIN {X 0,Y 736.028,Z 1154.105,A -85,B 0,C 180,E1 27801.327,E2 27801.327} C_VEL
LIN {X 0,Y 736.109,Z 1144.499,A -85,B 0,C 180,E1 27799.75,E2 27799.75} C_VEL
LIN {X 0,Y 736.179,Z 1133.698,A -85,B 0,C 180,E1 27798.165,E2 27798.165} C_VEL
LIN {X 0,Y 736.339,Z 1120.362,A -85,B 0,C 180,E1 27796.413,E2 27796.413} C_VEL
LIN {X 0,Y 736.514,Z 1103.727,A -85,B 0,C 180,E1 27794.488,E2 27794.488} C_VEL
LIN {X 0,Y 736.681,Z 1088.9,A -85,B 0,C 180,E1 27792.952,E2 27792.952} C_VEL
LIN {X 0,Y 736.903,Z 1072.462,A -85,B 0,C 180,E1 27791.406,E2 27791.406} C_VEL
LIN {X 0,Y 737.211,Z 1051.447,A -85,B 0,C 180,E1 27789.641,E2 27789.641} C_VEL
LIN {X 0,Y 737.462,Z 1033.873,A -85,B 0,C 180,E1 27788.317,E2 27788.317} C_VEL
LIN {X 0,Y 737.775,Z 1015.004,A -85,B 0,C 180,E1 27787.026,E2 27787.026} C_VEL
LIN {X 0,Y 738.202,Z 990.139,A -85,B 0,C 180,E1 27785.514,E2 27785.514} C_VEL
LIN {X 0,Y 738.502,Z 969.593,A -85,B 0,C 180,E1 27784.411,E2 27784.411} C_VEL
LIN {X 0,Y 738.799,Z 949.719,A -85,B 0,C 180,E1 27783.457,E2 27783.457} C_VEL
LIN {X 0,Y 739.1,Z 928.602,A -85,B 0,C 180,E1 27782.557,E2 27782.557} C_VEL
LIN {X 0,Y 739.529,Z 901.88,A -85,B 0,C 180,E1 27781.581,E2 27781.581} C_VEL
LIN {X 0,Y 739.818,Z 875.726,A -85,B 0,C 180,E1 27780.789,E2 27780.789} C_VEL
LIN {X 0,Y 740.087,Z 849.261,A -85,B 0,C 180,E1 27780.151,E2 27780.151} C_VEL
LIN {X 0,Y 740.312,Z 822.217,A -85,B 0,C 180,E1 27779.66,E2 27779.66} C_VEL
LIN {X 0,Y 740.493,Z 779.419,A -85,B 0,C 180,E1 27779.129,E2 27779.129} C_VEL
LIN {X 0,Y 741.158,Z 553.282,A -85,B 0,C 180,E1 27776.437,E2 27776.437} C_VEL
LIN {X 0,Y 741.812,Z 347.504,A -85,B 0,C 180,E1 27773.902,E2 27773.902} C_VEL
LIN {X 0,Y 739.974,Z 340.493,A -85,B 0,C 180,E1 27773.664,E2 27773.664} C_VEL
LIN {X 0,Y 739.913,Z 331.904,A -85,B 0,C 180,E1 27773.067,E2 27773.067} C_VEL
LIN {X 0,Y 736.108,Z 322.724,A -85,B 0,C 180,E1 27772.144,E2 27772.144} C_VEL
LIN {X 0,Y 736.084,Z 322.544,A -85,B 0,C 180,E1 27769.287,E2 27769.287} C_VEL
LIN {X 0,Y 736.064,Z 322.541,A -85,B 0,C 180,E1 27766.471,E2 27766.471} C_VEL
LIN {X 0,Y 736.096,Z 322.534,A -85,B 0,C 180,E1 27763.614,E2 27763.614} C_VEL
LIN {X 0,Y 736.082,Z 322.544,A -85,B 0,C 180,E1 27760.695,E2 27760.695} C_VEL
LIN {X 0,Y 736.074,Z 322.534,A -85,B 0,C 180,E1 27757.781,E2 27757.781} C_VEL
LIN {X 0,Y 736.096,Z 322.545,A -85,B 0,C 180,E1 27754.734,E2 27754.734} C_VEL
LIN {X 0,Y 736.053,Z 322.537,A -85,B 0,C 180,E1 27751.895,E2 27751.895} C_VEL
LIN {X 0,Y 736.094,Z 322.537,A -85,B 0,C 180,E1 27749.098,E2 27749.098} C_VEL
LIN {X 0,Y 736.052,Z 322.536,A -85,B 0,C 180,E1 27746.2,E2 27746.2} C_VEL
LIN {X 0,Y 736.062,Z 322.536,A -85,B 0,C 180,E1 27743.455,E2 27743.455} C_VEL
LIN {X 0,Y 736.078,Z 322.537,A -85,B 0,C 180,E1 27740.399,E2 27740.399} C_VEL
LIN {X 0,Y 736.035,Z 322.539,A -85,B 0,C 180,E1 27737.716,E2 27737.716} C_VEL
LIN {X 0,Y 736.09,Z 322.533,A -85,B 0,C 180,E1 27734.957,E2 27734.957} C_VEL
LIN {X 0,Y 736.045,Z 322.541,A -85,B 0,C 180,E1 27731.996,E2 27731.996} C_VEL
LIN {X 0,Y 736.027,Z 322.539,A -85,B 0,C 180,E1 27729.461,E2 27729.461} C_VEL
LIN {X 0,Y 736.092,Z 322.537,A -85,B 0,C 180,E1 27726.709,E2 27726.709} C_VEL
LIN {X 0,Y 736.035,Z 322.543,A -85,B 0,C 180,E1 27723.817,E2 27723.817} C_VEL
LIN {X 0,Y 736.017,Z 322.539,A -85,B 0,C 180,E1 27721.323,E2 27721.323} C_VEL
LIN {X 0,Y 736.053,Z 322.539,A -85,B 0,C 180,E1 27718.755,E2 27718.755} C_VEL
LIN {X 0,Y 736.033,Z 322.542,A -85,B 0,C 180,E1 27715.715,E2 27715.715} C_VEL
LIN {X 0,Y 736.007,Z 322.543,A -85,B 0,C 180,E1 27713.254,E2 27713.254} C_VEL
LIN {X 0,Y 736.008,Z 322.541,A -85,B 0,C 180,E1 27710.933,E2 27710.933} C_VEL
LIN {X 0,Y 736.097,Z 322.542,A -85,B 0,C 180,E1 27708.164,E2 27708.164} C_VEL
LIN {X 0,Y 736.004,Z 322.541,A -85,B 0,C 180,E1 27705.3,E2 27705.3} C_VEL
LIN {X 0,Y 735.993,Z 322.544,A -85,B 0,C 180,E1 27703.017,E2 27703.017} C_VEL
LIN {X 0,Y 735.995,Z 322.539,A -85,B 0,C 180,E1 27700.723,E2 27700.723} C_VEL
LIN {X 0,Y 736.081,Z 322.542,A -85,B 0,C 180,E1 27697.981,E2 27697.981} C_VEL
LIN {X 0,Y 735.998,Z 322.537,A -85,B 0,C 180,E1 27695.162,E2 27695.162} C_VEL
LIN {X 0,Y 735.989,Z 322.545,A -85,B 0,C 180,E1 27692.84,E2 27692.84} C_VEL
LIN {X 0,Y 735.995,Z 322.544,A -85,B 0,C 180,E1 27690.541,E2 27690.541} C_VEL
LIN {X 0,Y 736.052,Z 322.543,A -85,B 0,C 180,E1 27687.958,E2 27687.958} C_VEL
LIN {X 0,Y 736.018,Z 322.544,A -85,B 0,C 180,E1 27685.002,E2 27685.002} C_VEL
LIN {X 0,Y 736.004,Z 322.544,A -85,B 0,C 180,E1 27682.608,E2 27682.608} C_VEL
LIN {X 0,Y 736.012,Z 322.546,A -85,B 0,C 180,E1 27680.257,E2 27680.257} C_VEL
LIN {X 0,Y 736.1,Z 322.543,A -85,B 0,C 180,E1 27677.432,E2 27677.432} C_VEL
LIN {X 0,Y 736.02,Z 322.549,A -85,B 0,C 180,E1 27674.613,E2 27674.613} C_VEL
LIN {X 0,Y 736.042,Z 322.748,A -85,B 0,C 180,E1 27674.476,E2 27674.476} C_VEL
LIN {X 0,Y 737.279,Z 325.966,A -85,B 0,C 180,E1 27674.157,E2 27674.157} C_VEL
LIN {X 0,Y 740.205,Z 332.359,A -85,B 0,C 180,E1 27673.498,E2 27673.498} C_VEL
LIN {X 0,Y 740.195,Z 351.283,A -85,B 0,C 180,E1 27672.246,E2 27672.246} C_VEL
LIN {X 0,Y 741.797,Z 358.005,A -85,B 0,C 180,E1 27672.047,E2 27672.047} C_VEL
LIN {X 0,Y 741.142,Z 568.487,A -85,B 0,C 180,E1 27669.455,E2 27669.455} C_VEL
LIN {X 0,Y 740.483,Z 793.823,A -85,B 0,C 180,E1 27666.775,E2 27666.775} C_VEL
LIN {X 0,Y 740.313,Z 833.203,A -85,B 0,C 180,E1 27666.281,E2 27666.281} C_VEL
LIN {X 0,Y 740.078,Z 859.861,A -85,B 0,C 180,E1 27665.791,E2 27665.791} C_VEL
LIN {X 0,Y 739.824,Z 885.812,A -85,B 0,C 180,E1 27665.164,E2 27665.164} C_VEL
LIN {X 0,Y 739.517,Z 913.602,A -85,B 0,C 180,E1 27664.32,E2 27664.32} C_VEL
LIN {X 0,Y 739.092,Z 939.466,A -85,B 0,C 180,E1 27663.363,E2 27663.363} C_VEL
LIN {X 0,Y 738.79,Z 960.675,A -85,B 0,C 180,E1 27662.454,E2 27662.454} C_VEL
LIN {X 0,Y 738.489,Z 981.246,A -85,B 0,C 180,E1 27661.46,E2 27661.46} C_VEL
LIN {X 0,Y 738.111,Z 1005.682,A -85,B 0,C 180,E1 27660.126,E2 27660.126} C_VEL
LIN {X 0,Y 737.733,Z 1026.897,A -85,B 0,C 180,E1 27658.805,E2 27658.805} C_VEL
LIN {X 0,Y 737.448,Z 1045.341,A -85,B 0,C 180,E1 27657.532,E2 27657.532} C_VEL
LIN {X 0,Y 737.182,Z 1066.23,A -85,B 0,C 180,E1 27655.937,E2 27655.937} C_VEL
LIN {X 0,Y 736.851,Z 1085.146,A -85,B 0,C 180,E1 27654.305,E2 27654.305} C_VEL
LIN {X 0,Y 736.68,Z 1100.568,A -85,B 0,C 180,E1 27652.838,E2 27652.838} C_VEL
LIN {X 0,Y 736.469,Z 1117.984,A -85,B 0,C 180,E1 27651.004,E2 27651.004} C_VEL
LIN {X 0,Y 736.294,Z 1132.508,A -85,B 0,C 180,E1 27649.268,E2 27649.268} C_VEL
LIN {X 0,Y 736.197,Z 1144.249,A -85,B 0,C 180,E1 27647.712,E2 27647.712} C_VEL
LIN {X 0,Y 736.09,Z 1154.735,A -85,B 0,C 180,E1 27646.169,E2 27646.169} C_VEL
LIN {X 0,Y 736.043,Z 1164.522,A -85,B 0,C 180,E1 27644.555,E2 27644.555} C_VEL
LIN {X 0,Y 735.988,Z 1174.753,A -85,B 0,C 180,E1 27642.635,E2 27642.635} C_VEL
LIN {X 0,Y 735.949,Z 1184.911,A -85,B 0,C 180,E1 27640.331,E2 27640.331} C_VEL
LIN {X 0,Y 735.928,Z 1192.135,A -85,B 0,C 180,E1 27638.281,E2 27638.281} C_VEL
LIN {X 0,Y 735.918,Z 1197.734,A -85,B 0,C 180,E1 27636.24,E2 27636.24} C_VEL
LIN {X 0,Y 735.912,Z 1201.927,A -85,B 0,C 180,E1 27634.052,E2 27634.052} C_VEL
LIN {X 0,Y 735.912,Z 1204.212,A -85,B 0,C 180,E1 27632.025,E2 27632.025} C_VEL
LIN {X 0,Y 735.898,Z 1204.939,A -85,B 0,C 180,E1 27629.767,E2 27629.767} C_VEL
LIN {X 0,Y 735.908,Z 1203.976,A -85,B 0,C 180,E1 27627.664,E2 27627.664} C_VEL
LIN {X 0,Y 735.91,Z 1201.304,A -85,B 0,C 180,E1 27625.559,E2 27625.559} C_VEL
LIN {X 0,Y 735.92,Z 1197.153,A -85,B 0,C 180,E1 27623.525,E2 27623.525} C_VEL
LIN {X 0,Y 735.931,Z 1191.152,A -85,B 0,C 180,E1 27621.405,E2 27621.405} C_VEL
LIN {X 0,Y 735.931,Z 1183.319,A -85,B 0,C 180,E1 27619.273,E2 27619.273} C_VEL
LIN {X 0,Y 735.999,Z 1173.526,A -85,B 0,C 180,E1 27617.127,E2 27617.127} C_VEL
LIN {X 0,Y 736.045,Z 1164.527,A -85,B 0,C 180,E1 27615.445,E2 27615.445} C_VEL
LIN {X 0,Y 736.092,Z 1154.646,A -85,B 0,C 180,E1 27613.817,E2 27613.817} C_VEL
LIN {X 0,Y 736.198,Z 1143.672,A -85,B 0,C 180,E1 27612.207,E2 27612.207} C_VEL
LIN {X 0,Y 736.364,Z 1129.29,A -85,B 0,C 180,E1 27610.322,E2 27610.322} C_VEL
LIN {X 0,Y 736.522,Z 1112.619,A -85,B 0,C 180,E1 27608.414,E2 27608.414} C_VEL
LIN {X 0,Y 736.685,Z 1097.977,A -85,B 0,C 180,E1 27606.906,E2 27606.906} C_VEL
LIN {X 0,Y 736.986,Z 1079.518,A -85,B 0,C 180,E1 27605.184,E2 27605.184} C_VEL
LIN {X 0,Y 737.229,Z 1060.165,A -85,B 0,C 180,E1 27603.586,E2 27603.586} C_VEL
LIN {X 0,Y 737.478,Z 1042.501,A -85,B 0,C 180,E1 27602.263,E2 27602.263} C_VEL
LIN {X 0,Y 737.894,Z 1020.413,A -85,B 0,C 180,E1 27600.77,E2 27600.77} C_VEL
LIN {X 0,Y 738.22,Z 997.837,A -85,B 0,C 180,E1 27599.43,E2 27599.43} C_VEL
LIN {X 0,Y 738.518,Z 977.727,A -85,B 0,C 180,E1 27598.361,E2 27598.361} C_VEL
LIN {X 0,Y 738.841,Z 956.618,A -85,B 0,C 180,E1 27597.36,E2 27597.36} C_VEL
LIN {X 0,Y 739.294,Z 929.675,A -85,B 0,C 180,E1 27596.257,E2 27596.257} C_VEL
LIN {X 0,Y 739.567,Z 907.043,A -85,B 0,C 180,E1 27595.472,E2 27595.472} C_VEL
LIN {X 0,Y 739.849,Z 883.67,A -85,B 0,C 180,E1 27594.779,E2 27594.779} C_VEL
LIN {X 0,Y 740.115,Z 856.87,A -85,B 0,C 180,E1 27594.145,E2 27594.145} C_VEL
LIN {X 0,Y 740.323,Z 829.686,A -85,B 0,C 180,E1 27593.667,E2 27593.667} C_VEL
LIN {X 0,Y 740.663,Z 729.101,A -85,B 0,C 180,E1 27592.464,E2 27592.464} C_VEL
LIN {X 0,Y 741.342,Z 506.164,A -85,B 0,C 180,E1 27589.788,E2 27589.788} C_VEL
LIN {X 0,Y 741.643,Z 356.641,A -85,B 0,C 180,E1 27587.924,E2 27587.924} C_VEL
LIN {X 0,Y 740.052,Z 350.368,A -85,B 0,C 180,E1 27587.714,E2 27587.714} C_VEL
LIN {X 0,Y 740.205,Z 332.359,A -85,B 0,C 180,E1 27586.502,E2 27586.502} C_VEL
LIN {X 0,Y 736.094,Z 323.047,A -85,B 0,C 180,E1 27585.549,E2 27585.549} C_VEL
LIN {X 0,Y 736.017,Z 322.549,A -85,B 0,C 180,E1 27585.495,E2 27585.495} C_VEL
LIN {X 0,Y 736.081,Z 322.544,A -85,B 0,C 180,E1 27582.781,E2 27582.781} C_VEL
LIN {X 0,Y 736.024,Z 322.545,A -85,B 0,C 180,E1 27579.867,E2 27579.867} C_VEL
LIN {X 0,Y 736.006,Z 322.543,A -85,B 0,C 180,E1 27577.49,E2 27577.49} C_VEL
LIN {X 0,Y 736.011,Z 322.542,A -85,B 0,C 180,E1 27575.133,E2 27575.133} C_VEL
LIN {X 0,Y 736.099,Z 322.543,A -85,B 0,C 180,E1 27572.265,E2 27572.265} C_VEL
LIN {X 0,Y 736.007,Z 322.544,A -85,B 0,C 180,E1 27569.548,E2 27569.548} C_VEL
LIN {X 0,Y 735.995,Z 322.542,A -85,B 0,C 180,E1 27567.248,E2 27567.248} C_VEL
LIN {X 0,Y 736,Z 322.542,A -85,B 0,C 180,E1 27564.907,E2 27564.907} C_VEL
LIN {X 0,Y 736.1,Z 322.538,A -85,B 0,C 180,E1 27562.103,E2 27562.103} C_VEL
LIN {X 0,Y 735.995,Z 322.545,A -85,B 0,C 180,E1 27559.277,E2 27559.277} C_VEL
LIN {X 0,Y 735.984,Z 322.54,A -85,B 0,C 180,E1 27556.978,E2 27556.978} C_VEL
LIN {X 0,Y 735.989,Z 322.544,A -85,B 0,C 180,E1 27554.698,E2 27554.698} C_VEL
LIN {X 0,Y 736.071,Z 322.543,A -85,B 0,C 180,E1 27551.996,E2 27551.996} C_VEL
LIN {X 0,Y 736.003,Z 322.544,A -85,B 0,C 180,E1 27549.146,E2 27549.146} C_VEL
LIN {X 0,Y 735.991,Z 322.541,A -85,B 0,C 180,E1 27546.788,E2 27546.788} C_VEL
LIN {X 0,Y 735.997,Z 322.541,A -85,B 0,C 180,E1 27544.519,E2 27544.519} C_VEL
LIN {X 0,Y 736.048,Z 322.545,A -85,B 0,C 180,E1 27541.946,E2 27541.946} C_VEL
LIN {X 0,Y 736.021,Z 322.541,A -85,B 0,C 180,E1 27538.971,E2 27538.971} C_VEL
